	16#4401:
		CreateDriveErrMsgDetails := enumMotorEvents.MotorGeneralError;
		fnLogMsg(ADR(LogMsg_0),LOG_ERROR,'BeckHoff Drive ErrorId %d Starttype not supported',UDINT_TO_DINT(ErrorId),0,0);
	16#4402:
		CreateDriveErrMsgDetails := enumMotorEvents.MotorGeneralError;
		fnLogMsg(ADR(LogMsg_0),LOG_ERROR,'BeckHoff Drive ErrorId %d Command rejected',UDINT_TO_DINT(ErrorId),0,0);
	16#4405:
		CreateDriveErrMsgDetails := enumMotorEvents.MotorGeneralError;
		fnLogMsg(ADR(LogMsg_0),LOG_ERROR,'BeckHoff Drive ErrorId %d Invalid modulo subtype',UDINT_TO_DINT(ErrorId),0,0);
	16#4410:
		CreateDriveErrMsgDetails := enumMotorEvents.MotorGeneralError;
		fnLogMsg(ADR(LogMsg_0),LOG_ERROR,'BeckHoff Drive ErrorId %d Target overrun',UDINT_TO_DINT(ErrorId),0,0);
	16#4411:
		CreateDriveErrMsgDetails := enumMotorEvents.MotorSupplyError;
		fnLogMsg(ADR(LogMsg_0),LOG_ERROR,'BeckHoff Drive ErrorId %d DC-Link undervoltage',UDINT_TO_DINT(ErrorId),0,0);
	16#4412:
 		CreateDriveErrMsgDetails := enumMotorEvents.MotorSupplyError;
		fnLogMsg(ADR(LogMsg_0),LOG_ERROR,'BeckHoff Drive ErrorId %d 2 DC-Link overvoltage',UDINT_TO_DINT(ErrorId),0,0);
	16#4413: 
		CreateDriveErrMsgDetails := enumMotorEvents.MotorSupplyError;
		fnLogMsg(ADR(LogMsg_0),LOG_ERROR,'BeckHoff Drive ErrorId %d I2T Amplifier overload',UDINT_TO_DINT(ErrorId),0,0);
	16#4414:
		CreateDriveErrMsgDetails := enumMotorEvents.MotorSupplyError;
		fnLogMsg(ADR(LogMsg_0),LOG_ERROR,'BeckHoff Drive ErrorId %d I2T Motor overload',UDINT_TO_DINT(ErrorId),0,0);
	16#4415:
		CreateDriveErrMsgDetails := enumMotorEvents.MotorSpeedError;
		fnLogMsg(ADR(LogMsg_0),LOG_ERROR,'BeckHoff Drive ErrorId %d Speed limitation active',UDINT_TO_DINT(ErrorId),0,0);
	16#4416:
		CreateDriveErrMsgDetails := enumMotorEvents.MotorPositionError;
		fnLogMsg(ADR(LogMsg_0),LOG_ERROR,'BeckHoff Drive ErrorId %d Step lost detected',UDINT_TO_DINT(ErrorId),0,0);
	16#8001:
		CreateDriveErrMsgDetails := enumMotorEvents.MotorGeneralError;
		fnLogMsg(ADR(LogMsg_0),LOG_ERROR,'BeckHoff Drive ErrorId %d Error',UDINT_TO_DINT(ErrorId),0,0);
	16#8002:
		CreateDriveErrMsgDetails := enumMotorEvents.DriveComError ;
		fnLogMsg(ADR(LogMsg_0),LOG_ERROR,'BeckHoff Drive ErrorId %d Communication aborted',UDINT_TO_DINT(ErrorId),0,0);

	16#8003:
		CreateDriveErrMsgDetails := enumMotorEvents.PLCIllegalParam;
		fnLogMsg(ADR(LogMsg_0),LOG_ERROR,'BeckHoff Drive ErrorId %d Configuration error',UDINT_TO_DINT(ErrorId),0,0);
	16#8100:
		CreateDriveErrMsgDetails := enumMotorEvents.MotorGeneralError;
		fnLogMsg(ADR(LogMsg_0),LOG_ERROR,'BeckHoff Drive ErrorId %d Status word set',UDINT_TO_DINT(ErrorId),0,0);
	16#8101:
		CreateDriveErrMsgDetails := enumMotorEvents.PLCIllegalParam;
		fnLogMsg(ADR(LogMsg_0),LOG_ERROR,'BeckHoff Drive ErrorId %d Operation mode incompatible to PDO',UDINT_TO_DINT(ErrorId),0,0);
	16#8102:
		CreateDriveErrMsgDetails := enumMotorEvents.PLCIllegalParam;
		fnLogMsg(ADR(LogMsg_0),LOG_ERROR,'BeckHoff Drive ErrorId %d Invalid combination of Inputs and Outputs PDOs',UDINT_TO_DINT(ErrorId),0,0);

	16#8104:
		CreateDriveErrMsgDetails := enumMotorEvents.MotorOverTemp ;
		fnLogMsg(ADR(LogMsg_0),LOG_ERROR,'BeckHoff Drive ErrorId %d Terminal-Overtemperature',UDINT_TO_DINT(ErrorId),0,0);
	
	16#8105:
		CreateDriveErrMsgDetails := enumMotorEvents.MotorGeneralError ;
		fnLogMsg(ADR(LogMsg_0),LOG_ERROR,'BeckHoff Drive ErrorId %d PD-Watchdog',UDINT_TO_DINT(ErrorId),0,0);
	16#8135:
		CreateDriveErrMsgDetails := enumMotorEvents.MotorGeneralError ;
		fnLogMsg(ADR(LogMsg_0),LOG_ERROR,'BeckHoff Drive ErrorId %d Large cycle time',UDINT_TO_DINT(ErrorId),0,0);
	16#8200:
		CreateDriveErrMsgDetails := enumMotorEvents.PLCillegalMsg ;
		fnLogMsg(ADR(LogMsg_0),LOG_ERROR,'BeckHoff Drive ErrorId %d Write access error',UDINT_TO_DINT(ErrorId),0,0);
	16#8201:
		CreateDriveErrMsgDetails := enumMotorEvents.MotorSupplyError ;
		fnLogMsg(ADR(LogMsg_0),LOG_ERROR,'BeckHoff Drive ErrorId %d No com to field-side (Auxiliary voltage missing)',UDINT_TO_DINT(ErrorId),0,0);
	16#82FF:
		CreateDriveErrMsgDetails := enumMotorEvents.MotorGeneralError ;
		fnLogMsg(ADR(LogMsg_0),LOG_ERROR,'BeckHoff Drive ErrorId %d Bootmode not activated',UDINT_TO_DINT(ErrorId),0,0);
	16#8300:
		CreateDriveErrMsgDetails := enumMotorEvents.MotorPositionError ;
		fnLogMsg(ADR(LogMsg_0),LOG_ERROR,'BeckHoff Drive ErrorId %d Set position error',UDINT_TO_DINT(ErrorId),0,0);
	16#8301:
		CreateDriveErrMsgDetails := enumMotorEvents.PLCIllegalParam ;
		fnLogMsg(ADR(LogMsg_0),LOG_ERROR,'BeckHoff Drive ErrorId %d Encoder increments not configured',UDINT_TO_DINT(ErrorId),0,0);
	16#8302:
		CreateDriveErrMsgDetails := enumMotorEvents.MotorFeedBackErr ;
		fnLogMsg(ADR(LogMsg_0),LOG_ERROR,'BeckHoff Drive ErrorId %d Encoder-Error',UDINT_TO_DINT(ErrorId),0,0);

	16#8400:
		CreateDriveErrMsgDetails := enumMotorEvents.PLCIllegalParam;
		fnLogMsg(ADR(LogMsg_0),LOG_ERROR,'BeckHoff Drive ErrorId %d Incorrect drive configuration',UDINT_TO_DINT(ErrorId),0,0);
		
	16#8401:
		CreateDriveErrMsgDetails := enumMotorEvents.MotorSpeedError;
		fnLogMsg(ADR(LogMsg_0),LOG_ERROR,'BeckHoff Drive ErrorId %d Limiting of calibration velocity',UDINT_TO_DINT(ErrorId),0,0);
		
	16#8402:
		CreateDriveErrMsgDetails := enumMotorEvents.DriveNotEnabled;
		fnLogMsg(ADR(LogMsg_0),LOG_ERROR,'BeckHoff Drive ErrorId %d Emergency stop activated',UDINT_TO_DINT(ErrorId),0,0);
	16#8403:
		CreateDriveErrMsgDetails := enumMotorEvents.MotorSupplyError;
		fnLogMsg(ADR(LogMsg_0),LOG_ERROR,'BeckHoff Drive ErrorId %d ADC Error',UDINT_TO_DINT(ErrorId),0,0);
	16#8404:
		CreateDriveErrMsgDetails := enumMotorEvents.MotorSupplyError;
		fnLogMsg(ADR(LogMsg_0),LOG_ERROR,'BeckHoff Drive ErrorId %d Overcurrent',UDINT_TO_DINT(ErrorId),0,0);
	16#8405:
		CreateDriveErrMsgDetails := enumMotorEvents.MotorPositionError;
		fnLogMsg(ADR(LogMsg_0),LOG_ERROR,'BeckHoff Drive ErrorId %d Invalid modulo position',UDINT_TO_DINT(ErrorId),0,0);
	16#8406:
		CreateDriveErrMsgDetails := enumMotorEvents.MotorSupplyError;
		fnLogMsg(ADR(LogMsg_0),LOG_ERROR,'BeckHoff Drive ErrorId %d Undervoltage DC-Link',UDINT_TO_DINT(ErrorId),0,0);
	16#8407:
		CreateDriveErrMsgDetails := enumMotorEvents.MotorSupplyError;
		fnLogMsg(ADR(LogMsg_0),LOG_ERROR,'BeckHoff Drive ErrorId %d Overvoltage DC-Link',UDINT_TO_DINT(ErrorId),0,0);
	16#8408:
		CreateDriveErrMsgDetails := enumMotorEvents.MotorSupplyError;
		fnLogMsg(ADR(LogMsg_0),LOG_ERROR,'BeckHoff Drive ErrorId %d I2T-Model Amplifier overload',UDINT_TO_DINT(ErrorId),0,0);
	16#8409:
		CreateDriveErrMsgDetails := enumMotorEvents.MotorSupplyError;
		fnLogMsg(ADR(LogMsg_0),LOG_ERROR,'BeckHoff Drive ErrorId %d I2T-Model motor overload',UDINT_TO_DINT(ErrorId),0,0);
		
	16#8415:
		CreateDriveErrMsgDetails := enumMotorEvents.PLCIllegalParam;
		fnLogMsg(ADR(LogMsg_0),LOG_ERROR,'BeckHoff Drive ErrorId %d Invalid modulo factor',UDINT_TO_DINT(ErrorId),0,0);
	16#8440:
		CreateDriveErrMsgDetails := enumMotorEvents.MotorSupplyError;
		fnLogMsg(ADR(LogMsg_0),LOG_ERROR,'BeckHoff Drive ErrorId %d Motor cable not connected',UDINT_TO_DINT(ErrorId),0,0);

	ELSE
		fnLogMsg(ADR(LogMsg_0),LOG_ERROR,'unknown BeckHoff Drive ErrorId %d ',UDINT_TO_DINT(ErrorId),0,0);
		CreateDriveErrMsgDetails := enumMotorEvents.NoEvents;
END_CASE
END_METHOD

METHOD DriveErrorHandling : BOOL
VAR_INST
	
	ErrHandleState	: INT;

	SoEReset_FB	: FB_SoEReset;
	EcSoERead_DriveError_FB		: FB_EcSoERead;
	tmpDriveErrId				: UINT;
	NewMsgID					: BYTE;
	PrevMsgID					: BYTE;
	DiagMsg                     : STRING[100];
	EcCoeSdoRead_DriveErrorFB	: FB_EcCoeSdoRead;
	MC_Reset_FB					: MC_Reset;
	tempErrorEntry			    : Eh_ErrorEntry_typ;
	ErrorByte1                  : UINT;
	ErrorByte2                  : UINT;
	BeckHoffLastError       	: UDINT; 
	BeckHoffLastErrorCounter    : UDINT := 0; 
END_VAR


CASE ErrHandleState OF
	0: // logic init
		GetErrCanAdr();	
		ErrHandleState	:= 200;
		
		
	//************************* CAN Logic **********************************************
	200: // wait errors
		{warning disable C0371}
		IF AxisRef.Status.DriveDeviceError OR AxisRef.NcToPlc.ErrorCode = 18000 THEN
			SoEReset_FB.Execute				:= FALSE;
			EcSoERead_DriveError_FB.bExecute	:= FALSE;
			ErrHandleState	:= 210;
		ELSIF AxisRef.NcToPlc.ErrorCode <> 0 
			AND AxisRef.NcToPlc.ErrorCode <> 18000 THEN
			// ETZ Axis.NcToPlc.ErrorCode
			ErrHandleState	:= 300;
		ELSIF AxisCtrlPtr^.Output.Error.fbErrorHandler.EntriesCount > 0 THEN
			// do nothing
		END_IF
		
		IF AxisRef.Status.DriveDeviceError = FALSE THEN
			BeckHoffLastError := 0;
			BeckHoffLastErrorCounter := 0;
		END_IF
		{warning restore C0371}
	210: // wait speed decrease
		IF AxisCtrlPtr^.Output.monitor.ActVelocity < 500 THEN
			ErrHandleState	:= 211;	// read can error
		END_IF
		
	211:// MSG ID read new 
		PrevMsgID := NewMsgID;
		EcCoeSdoRead_DriveErrorFB.sNetId		:= strEcNetId;
		EcCoeSdoRead_DriveErrorFB.nSlaveAddr	:= AxisCtrlPtr^.Input.Parameter.Drive.EtherCatAddr;
		CoeErrIdSubIndex					    := 16#02 ; 			// MSG ID read new 
		EcCoeSdoRead_DriveErrorFB.nIndex		:= CoeErrIdIndex; 
		EcCoeSdoRead_DriveErrorFB.nSubIndex	    := CoeErrIdSubIndex; 
		EcCoeSdoRead_DriveErrorFB.pDstBuf		:= ADR(NewMsgID);
		EcCoeSdoRead_DriveErrorFB.cbBufLen		:= SIZEOF(NewMsgID);
		EcCoeSdoRead_DriveErrorFB.tTimeout		:= T#10S;
		IF NOT EcCoeSdoRead_DriveErrorFB.bBusy THEN
			EcCoeSdoRead_DriveErrorFB.bExecute		:= TRUE;
			
			ErrHandleState	:= 212;
		END_IF	
	212:
		IF NOT EcCoeSdoRead_DriveErrorFB.bBusy THEN
			EcCoeSdoRead_DriveErrorFB.bExecute		:= FALSE;
			IF NOT EcCoeSdoRead_DriveErrorFB.bError THEN				
				
				IF PrevMsgID <> NewMsgID THEN
					// Read Msg
					ErrHandleState	:= 213;
				ELSE
					ErrHandleState	:= 200;	
				END_IF
			ELSE
				fnLogMsg(ADR(LogMsg_0),LOG_ERROR,'NO LINKS FOR DRIVE or Wrong Obj  obj index=%d subindex=%d ErrID %d ',CoeErrIdIndex,CoeErrIdSubIndex,UDINT_TO_DINT(EcCoeSdoRead_DriveErrorFB.nErrId ));
				ErrHandleState	:= 221;	
				DebugError := 1;
			END_IF
		END_IF
	213:
		EcCoeSdoRead_DriveErrorFB.sNetId		:= strEcNetId;
		EcCoeSdoRead_DriveErrorFB.nSlaveAddr	:= AxisCtrlPtr^.Input.Parameter.Drive.EtherCatAddr;
		
		CoeErrIdSubIndex					    := NewMsgID ; 	
		
		EcCoeSdoRead_DriveErrorFB.nIndex		:= CoeErrIdIndex; 
		EcCoeSdoRead_DriveErrorFB.nSubIndex	    := CoeErrIdSubIndex; 
		EcCoeSdoRead_DriveErrorFB.pDstBuf		:= ADR(DiagMsg);
		EcCoeSdoRead_DriveErrorFB.cbBufLen		:= ErrorMSgSize;
		EcCoeSdoRead_DriveErrorFB.tTimeout		:= T#20S;
		IF NOT EcCoeSdoRead_DriveErrorFB.bBusy THEN
			EcCoeSdoRead_DriveErrorFB.bExecute		:= TRUE;
			ErrHandleState	:= 214;	// MC_Reset
		END_IF	
	214:
		IF NOT EcCoeSdoRead_DriveErrorFB.bBusy THEN
			EcCoeSdoRead_DriveErrorFB.bExecute		:= FALSE;
			IF NOT EcCoeSdoRead_DriveErrorFB.bError THEN
				
				ErrHandleState	:= 220;	// Parse error ID
				ErrorByte1 := DiagMsg[6];
				ErrorByte2 := DiagMsg[7]; 
								
				tmpDriveErrId := ErrorByte1 OR SHL(ErrorByte2,8) ;				
				
			ELSE
				fnLogMsg(ADR(LogMsg_0),LOG_ERROR,'St 214 Error read obj index=%d subindex=%d ErrID %d ',CoeErrIdIndex,CoeErrIdSubIndex,TO_DINT(EcCoeSdoRead_DriveErrorFB.nErrId) );
				ErrHandleState	:= 221;	
				
				DebugError := 2;
			END_IF
		END_IF	
	//Parse error ID
	220:
				IF tmpDriveErrId <> 1 THEN
					// Add Drive Error to ErrorHandler
					tmp_ErrorEntry.ErrorId		:= tmpDriveErrId;
		//			IF BeckHoffLastError <>  tmp_ErrorEntry.ErrorId OR BeckHoffLastErrorCounter > 10  THEN
					
						
						tmp_ErrorEntry.ErrorText	:= AxisCtrlPtr^.Input.Parameter.ThreadName;
						tmp_ErrorEntry.ErrorText	:= CONCAT(tmp_ErrorEntry.ErrorText,'Beckhoff Drive ErrorID: ');
						tmp_ErrorEntry.ErrorText	:= CONCAT(tmp_ErrorEntry.ErrorText, UDINT_TO_STRING(tmp_ErrorEntry.ErrorId));
						tmp_ErrorEntry.ErrorText	:= CONCAT(tmp_ErrorEntry.ErrorText, ', Or 0x');
						tmp_ErrorEntry.ErrorText	:= CONCAT(tmp_ErrorEntry.ErrorText, UDINT_TO_HEX_STRING(tmp_ErrorEntry.ErrorId));
						
						tmp_ErrorEntry.MotorEvents  := CreateDriveErrMsgDetails(tmp_ErrorEntry.ErrorId);
						fnLogMsg(ADR(LogMsg_0),LOG_ERROR,tmp_ErrorEntry.ErrorText,0,0,0);
						//ETZ to Add method for Log			
						AxisCtrlPtr^.Output.Error.fbErrorHandler.ErrorPush(tmp_ErrorEntry);
						BeckHoffLastError := tmp_ErrorEntry.ErrorId;
						BeckHoffLastErrorCounter := 0;
			(*		ELSE
						BeckHoffLastErrorCounter := BeckHoffLastErrorCounter + 1;	
					END_IF	*)
				END_IF				
				ErrHandleState	:= 300;	// MC_Reset
		
 	221:
				
					// Add Drive Error to ErrorHandler
					tmp_ErrorEntry.ErrorId		:= 16#8002;
					tmp_ErrorEntry.ErrorText	:= AxisCtrlPtr^.Input.Parameter.ThreadName;
					tmp_ErrorEntry.ErrorText	:= CONCAT(tmp_ErrorEntry.ErrorText,' Drive ErrorID: ');
					tmp_ErrorEntry.ErrorText	:= CONCAT(tmp_ErrorEntry.ErrorText, UDINT_TO_STRING(tmp_ErrorEntry.ErrorId));
					tmp_ErrorEntry.ErrorText	:= CONCAT(tmp_ErrorEntry.ErrorText, ', Or 0x');
					tmp_ErrorEntry.ErrorText	:= CONCAT(tmp_ErrorEntry.ErrorText, UDINT_TO_HEX_STRING(tmp_ErrorEntry.ErrorId));
					
					tmp_ErrorEntry.MotorEvents  := CreateDriveErrMsgDetails(tmp_ErrorEntry.ErrorId);
					fnLogMsg(ADR(LogMsg_0),LOG_ERROR,tmp_ErrorEntry.ErrorText,0,0,0);
					//ETZ to Add method for Log			
					AxisCtrlPtr^.Output.Error.fbErrorHandler.ErrorPush(tmp_ErrorEntry);
								
				ErrHandleState	:= 300;	// MC_Reset
	300: // Run MC_Reset
		MC_Reset_FB.Execute	:= TRUE;
		ErrHandleState		:= 301;
	301:
		{warning disable C0371}
		IF MC_Reset_FB.Done 
			AND AxisRef.NcToPlc.ErrorCode = 0
			(*AND Axis.Status.DriveDeviceError = FALSE*) THEN
			MC_Reset_FB.Execute	:= FALSE;
	
			ErrHandleState	:= 0;
		ELSIF (MC_Reset_FB.Done AND AxisRef.NcToPlc.ErrorCode <> 0) THEN
			
			MC_Reset_FB.Execute	:= FALSE;	
			ErrHandleState		:= 300;	
	
		ELSIF MC_Reset_FB.Error THEN
			MC_Reset_FB.Execute	:= FALSE;
			// Add FB Error to ErrorHandler
			tmp_ErrorEntry.ErrorId		:= MC_Reset_FB.ErrorID;
			tmp_ErrorEntry.ErrorText	:= 'FB MC_Reset_FB ErrorID: ';
			tmp_ErrorEntry.ErrorText	:= CONCAT(tmp_ErrorEntry.ErrorText, UDINT_TO_STRING(tmp_ErrorEntry.ErrorId));
			AxisCtrlPtr^.Output.Error.fbErrorHandler.ErrorPush(tmp_ErrorEntry);
			
			ErrHandleState	:= 0;
		END_IF
		{warning restore C0371}
		IF (AxisCtrlPtr^.Output.Status.CommunicationError = TRUE) THEN
			MC_Reset_FB.Execute	:= FALSE;
			ErrHandleState		:= 400;	
		END_IF
	400:
		IF (AxisCtrlPtr^.Output.Status.CommunicationError = FALSE) THEN
			ErrHandleState	:= 300;	
		END_IF
			

END_CASE

EcSoERead_DriveError_FB();
EcCoeSdoRead_DriveErrorFB();
{warning disable C0371}
SoEReset_FB(Axis:= AxisRef);
MC_Reset_FB(Axis:= AxisRef);
	
{warning restore C0371}
END_METHOD

METHOD GetErrCanAdr : BOOL
VAR_INPUT
END_VAR

CoeErrIdIndex		:= 16#10F3;

		
//CoeErrIdIndex	:= 16#603F;
END_METHOD

END_FUNCTION_BLOCK

// ---- POUs/Lib/Motion/CanOpenAxis/BeckHoff/BeckHoffIntegratedAxis_FB.TcPOU
FUNCTION_BLOCK PUBLIC BeckHoffIntegratedAxis_FB EXTENDS BeckHoffBasicAxis_FB  
VAR_INPUT		
	io_SafetyState: 	BOOL;	
END_VAR

VAR_OUTPUT	
END_VAR

VAR
	 
	
END_VAR


CoEDrive_Ctrl_Adr.DCVoltage.Index 	 := 16#6079; 
CoEDrive_Ctrl_Adr.DCVoltage.SunIndex  := 0;
CoEDrive_Ctrl_Adr.DCVoltage.Size      := 4;

AxisCtrlPtr^.Input.Parameter.Drive.eDriveType := enumDriveType.eIntegratedBeckhoff;	
AxisCtrlPtr^.Input.Parameter.Drive.VendorNameID := eVendorNameID.Beckhoff;
	
 	
SUPER^(AxisRef:=AxisRef);

AxisCtrlPtr^.Output.Status.DriveEnable:=	io_SafetyState;

METHOD GetCanOpenAdr : BOOL
VAR_INPUT
END_VAR
    SUPER^.GetCanOpenAdr();	
	
	
	CoEDrive_Ctrl_Adr.DCVoltage.Index 	 := 16#9010; 
	CoEDrive_Ctrl_Adr.DCVoltage.SunIndex  := 12;
	CoEDrive_Ctrl_Adr.DCVoltage.Size      := 2;
END_METHOD

METHOD HomeLagError : BOOL
VAR_INPUT
	Execute: BOOL;
END_VAR

VAR_INST
	LagErrorState : INT;
	HomingLagErrorTrig: 		Trigger;
	io_TorqueLimitPersent_Mem:	UINT;
	PositionBias:				LREAL;	
END_VAR
Reset:= Execute;
IF HomeTrig.EDGEPOS(Reset) THEN
	Reset:=	FALSE;
	LagErrorState:=1;
	HomingActive:= 	TRUE ;
	AxisCtrlPtr^.Output.Status.MC_Home.Done:= FALSE ;
	fbMC_MoveVel.Execute:= FALSE ;
	fbMC_MoveRel.Execute:= FALSE ;
END_IF

IF Execute THEN
	CASE LagErrorState OF
		
		1:		
			io_TorqueLimitPersent_Mem:=	io_TorqueLimitPersent;							
			io_TorqueLimitPersent:=	AxisCtrlPtr^.Input.Parameter.HomeOptions.stLagErr.TorqueLimitPersent;				
			LagErrorState:= LagErrorState +1;
						 		
		2:	
			IF WriteNC_AxisBoolParam(MC_AxisParameter:=MC_AxisParameter.EnablePosLagMonitoring,ParamValue:=FALSE) THEN
				LagErrorState:= LagErrorState +1;	
			END_IF
																
		3: 										
			IF AxisCtrlPtr^.Input.Parameter.HomeOptions.stBasic.StartDirection = eHomeModeOption.eNEGATIVE THEN								
				fbMC_MoveVel.Direction:= 	MC_Negative_Direction;  					
			ELSIF AxisCtrlPtr^.Input.Parameter.HomeOptions.stBasic.StartDirection = eHomeModeOption.ePOSITIVE THEN								
				fbMC_MoveVel.Direction:= 	MC_Positive_Direction;										
			END_IF
			
			fbMC_MoveVel.Velocity:= AxisCtrlPtr^.Input.Parameter.HomeOptions.stBasic.SwitchVelo;
	
			fbMC_MoveVel.Execute:= 	TRUE ;
			
			LagErrorState:= LagErrorState + 1;
			
		4: 	
			IF (ABS(AxisCtrlPtr^.Output.monitor.ActLagError) > AxisCtrlPtr^.Input.Parameter.HomeOptions.stLagErr.LagErr) THEN
				LagErrorState:= LagErrorState + 1;	
			END_IF
		
		5:	
			IF Stop() THEN
				LagErrorState:= LagErrorState + 2;
				Delay(IN:=	FALSE);					
			END_IF
(*					
		6:	InternalPowerHandle:=	TRUE;
			AxisCtrlPtr^.Input.Command.Power:= FALSE;
			IF AxisCtrlPtr^.Output.Status.AxisStatus.Disabled THEN
				LagErrorState:= LagErrorState + 1;	
			END_IF
*)			
		7:	Delay(IN:=	TRUE,PT:=T#1S);		
			IF Delay.Q THEN
				Delay(IN:=FALSE);	
				LagErrorState:= LagErrorState +2;
			END_IF
(*	
		8:	InternalPowerHandle:=	FALSE;
			AxisCtrlPtr^.Input.Command.Power:= TRUE;
			
			IF (AxisCtrlPtr^.Output.Status.AxisStatus.Disabled = FALSE) THEN
				
				io_TorqueLimitPersent:=	io_TorqueLimitPersent_Mem;	
				LagErrorState:= LagErrorState + 1;	
			END_IF
*)						
		9: 	io_TorqueLimitPersent:=	io_TorqueLimitPersent_Mem;	
			IF AxisCtrlPtr^.Input.Parameter.HomeOptions.stBasic.StartDirection = eHomeModeOption.eNEGATIVE THEN													
				fbMC_MoveRel.Distance:=		AxisCtrlPtr^.Input.Parameter.HomeOptions.stLagErr.TriggerOffsetPos ;					
			ELSIF AxisCtrlPtr^.Input.Parameter.HomeOptions.stBasic.StartDirection = eHomeModeOption.ePOSITIVE THEN								
				fbMC_MoveRel.Distance:=		AxisCtrlPtr^.Input.Parameter.HomeOptions.stLagErr.TriggerOffsetPos*(-1) ;											
			END_IF
			fbMC_MoveRel.Velocity:= AxisCtrlPtr^.Input.Parameter.HomeOptions.stBasic.TriggerVelo;
			
			fbMC_MoveRel.Execute:= 	TRUE ;
			LagErrorState:= LagErrorState + 1;
	 		
					
		10:	
			IF fbMC_MoveRel.Done THEN
				AxisCtrlPtr^.Output.monitor.stAbsEncoder.BlockOffsetPosition := AxisCtrlPtr^.Output.monitor.ActPosition ;
				(*				
				fbMC_Home.HomingMode:= 	MC_Direct ;
				fbMC_Home.Position:= 	(AxisCtrlPtr^.Input.Parameter.HomeOptions.stBasic.HomeSetPos); 
				fbMC_Home.Execute:= 	TRUE;
				LagErrorState:= LagErrorState + 1;*)
				LagErrorState:= 100;
			END_IF
			
		11:	IF fbMC_Home.Done THEN			
				fbMC_Home.Execute:= 	FALSE;
				LagErrorState:= 100;	
			END_IF
																				
		100:			
			AxisCtrlPtr^.Input.Command.Home:= FALSE ;
			HomingActive:= 				FALSE;
			fbMC_Home.Execute:= 		FALSE;
			AxisCtrlPtr^.Output.Status.MC_Home.Done:= TRUE ;
			HomeLagError:=	TRUE;
			LagErrorState:= 0;		
	END_CASE

END_IF
 
			
fbMC_MoveVel.Acceleration  	:= AxisCtrlPtr^.Input.Parameter.HomeOptions.stBasic.Acc;  
fbMC_MoveVel.Deceleration  	:= AxisCtrlPtr^.Input.Parameter.HomeOptions.stBasic.Dcc;  
fbMC_MoveVel.Jerk			:= AxisCtrlPtr^.Input.Parameter.HomeOptions.stBasic.Jerk;
fbMC_MoveVel.Options		:= AxisCtrlPtr^.Input.Parameter.Options;
fbMC_MoveVel.BufferMode		:= AxisCtrlPtr^.Input.Parameter.BufferMode;

fbMC_MoveRel.Acceleration  	:= AxisCtrlPtr^.Input.Parameter.HomeOptions.stBasic.Acc; 
fbMC_MoveRel.Deceleration  	:= AxisCtrlPtr^.Input.Parameter.HomeOptions.stBasic.Dcc;
fbMC_MoveRel.Jerk			:= AxisCtrlPtr^.Input.Parameter.HomeOptions.stBasic.Jerk;
fbMC_MoveRel.Options		:= AxisCtrlPtr^.Input.Parameter.Options;
fbMC_MoveRel.BufferMode		:= AxisCtrlPtr^.Input.Parameter.BufferMode;

{warning disable C0371}
//Warning: Access to VAR_IN_OUT <Var> declared in <POU> from external context <Method/Transition/Property>

fbMC_Home(Axis:= AxisRef);	
fbMC_MoveVel(Axis:= AxisRef);
fbMC_MoveRel(Axis:= AxisRef);

fbMC_Stop.Deceleration:= 	AxisCtrlPtr^.Input.Parameter.Deceleration;
fbMC_Stop.Jerk:=			AxisCtrlPtr^.Input.Parameter.Jerk;
fbMC_Stop.Options:= 		AxisCtrlPtr^.Input.Parameter.Options;
fbMC_Stop(Axis := AxisRef) ;
{warning restore C0371}

THIS^.HomingGlobalHandle();
END_METHOD

METHOD ReadActualTorque : LREAL
VAR_INPUT
END_VAR
VAR_INST
		
END_VAR


// Units [rms]

{warning disable C0371}
IF AxisCtrlPtr^.Output.Status.Drive.ActiveHW THEN
	AxisCtrlPtr^.Output.monitor.ActualTorque	:=  ( -(AxisRef.NcToPlc.ActTorque) / 100.0) * AxisCtrlPtr^.Input.Parameter.Ratedtorque;
ELSE
	AxisCtrlPtr^.Output.monitor.ActualTorque	:=  ((THIS^.io_ActualTorque) / 1000.0) * AxisCtrlPtr^.Input.Parameter.Ratedtorque;
END_IF	

{warning restore C0371}
END_METHOD

END_FUNCTION_BLOCK

// ---- POUs/Lib/Motion/CanOpenAxis/BeckHoff/bk5xxxBasicAxis_FB.TcPOU
FUNCTION_BLOCK bk5xxxBasicAxis_FB EXTENDS BeckHoffBasicAxis_FB
VAR_INPUT
	pDigIn: 	POINTER TO INT;	
END_VAR
VAR_OUTPUT
END_VAR
VAR
	
END_VAR


AxisCtrlPtr^.Input.Parameter.Drive.eDriveType	:= enumDriveType.e5xxxBeckhoff;
AxisCtrlPtr^.Input.Parameter.Drive.VendorNameID	:= eVendorNameID.Beckhoff;


SUPER^(AxisRef:=AxisRef);

IF (pDigIn <> 0) THEN
	AxisCtrlPtr^.Output.Status.DriveEnable	:= pDigIn^.7;
ELSE
	AxisCtrlPtr^.Output.Status.DriveEnable	:= TRUE;
END_IF

END_FUNCTION_BLOCK

// ---- POUs/Lib/Motion/CanOpenAxis/BeckHoff/el7xxxBasicAxis_FB.TcPOU
FUNCTION_BLOCK el7xxxBasicAxis_FB EXTENDS BeckHoffBasicAxis_FB
VAR_INPUT
	pDigIn: 	POINTER TO INT;	
END_VAR
VAR_OUTPUT
END_VAR
VAR
	
END_VAR


AxisCtrlPtr^.Input.Parameter.Drive.eDriveType := enumDriveType.eEL70xx;
AxisCtrlPtr^.Input.Parameter.Drive.VendorNameID := eVendorNameID.Beckhoff;


SUPER^(AxisRef:=AxisRef);

IF (pDigIn <> 0) THEN
	AxisCtrlPtr^.Output.Status.DriveEnable	:= pDigIn^.7;
ELSE
	AxisCtrlPtr^.Output.Status.DriveEnable	:= TRUE;
END_IF

METHOD HomeLagErrExternFeedBack : BOOL
VAR_INPUT
	Execute: BOOL;
END_VAR

VAR_INST
	fbEcCoeSdoWriteMaxCurrent	: FB_EcCoeSdoWrite;
	State:INT;	
	ExtLagErrPrevState : INT;
	HomeTrig: Trigger;
	Reset:BOOL;	
	Delay:	TON;	
	LastActExternEncodPos:		UDINT;
	DiffExternEncodPos:			DINT;
	LatchSetPos:				LREAL;			
	CalckedLagError:			LREAL;
	EncdSampleTimer:			TON;
	StartPosMonitor:			BOOL;
		
END_VAR
Reset:= Execute;
IF HomeTrig.EDGEPOS(Reset) THEN
	Reset:=	FALSE;
	State:=1;
	
	HomeLagErrExternFeedBack:= FALSE ;
	HomingActive:= 	TRUE ;
	AxisCtrlPtr^.Output.Status.MC_Home.Done:= FALSE ;
	fbMC_MoveVel.Execute:= FALSE ;
	fbMC_MoveRel.Execute:= FALSE ;
END_IF

IF Execute THEN
	CASE State OF
		
		1:									
			fbEcCoeSdoWriteMaxCurrent.sNetId:= 		strEcNetId;
			fbEcCoeSdoWriteMaxCurrent.nSlaveAddr:= 	AxisCtrlPtr^.Input.Parameter.Drive.EtherCatAddr;
			fbEcCoeSdoWriteMaxCurrent.nSubIndex:=	1;
			fbEcCoeSdoWriteMaxCurrent.nIndex:= 		16#8010;  			
			fbEcCoeSdoWriteMaxCurrent.pSrcBuf:=		 ADR(AxisCtrlPtr^.Input.Parameter.HomeOptions.stLagErr.BlockSearchMaxCurrent); 
			fbEcCoeSdoWriteMaxCurrent.cbBufLen:= 	SIZEOF(AxisCtrlPtr^.Input.Parameter.HomeOptions.stLagErr.BlockSearchMaxCurrent); 
			fbEcCoeSdoWriteMaxCurrent.bExecute:= 	TRUE; 
			fbEcCoeSdoWriteMaxCurrent.tTimeout:= 	T#2S;					
			State:= State +1;							
			 
		2:		
			IF NOT fbEcCoeSdoWriteMaxCurrent.bBusy THEN
				fbEcCoeSdoWriteMaxCurrent.bExecute:= FALSE;
				IF NOT fbEcCoeSdoWriteMaxCurrent.bError THEN																									
					State:= State +1;
				ELSE
					fbEcCoeSdoWriteMaxCurrent.bExecute:= FALSE;
					fnLogMsg(ADR(LogMsg_0),LOG_ERROR,Concat('ADS Error Code %d: ',F_ADStoStr(fbEcCoeSdoWriteMaxCurrent.nErrId)),UDINT_TO_DINT(fbEcCoeSdoWriteMaxCurrent.nErrId),0,0);
					State:= 0;				
				END_IF				
			END_IF 		 
		3:	
			IF WriteNC_AxisBoolParam(MC_AxisParameter:=MC_AxisParameter.EnablePosLagMonitoring,ParamValue:=FALSE) THEN
				State:= State +1;	
			END_IF
						
										
		4: 										
			IF AxisCtrlPtr^.Input.Parameter.HomeOptions.stBasic.StartDirection = eHomeModeOption.eNEGATIVE THEN								
				fbMC_MoveVel.Direction:= 	MC_Negative_Direction; 					
			ELSIF AxisCtrlPtr^.Input.Parameter.HomeOptions.stBasic.StartDirection = eHomeModeOption.ePOSITIVE THEN								
				fbMC_MoveVel.Direction:= 	MC_Positive_Direction;										
			END_IF
			
			fbMC_MoveVel.Velocity:= AxisCtrlPtr^.Input.Parameter.HomeOptions.stBasic.SwitchVelo;			
			fbMC_MoveVel.Execute:= 	TRUE ;
			LastActExternEncodPos:=	AxisCtrlPtr^.Output.monitor.ActExternEncodPos;						
			State:= State + 1;
			
		5:	IF AxisCtrlPtr^.Output.Status.AxisStatus.ContinuousMotion THEN
				EncdSampleTimer(IN:= NOT(EncdSampleTimer.Q),PT:=T#0.2S);
				IF EncdSampleTimer.Q THEN	
					State:= State + 1;
				END_IF	
			END_IF
		6: 							
			DiffExternEncodPos:=ABS(UDINT_TO_DINT(AxisCtrlPtr^.Output.monitor.ActExternEncodPos) - UDINT_TO_DINT(LastActExternEncodPos));
			IF DiffExternEncodPos <= 4 THEN
				LatchSetPos:=	AxisCtrlPtr^.Output.monitor.ActPosition;			
				State:= State + 1;
			ELSE
				LastActExternEncodPos:=	AxisCtrlPtr^.Output.monitor.ActExternEncodPos;	
				State:= 5;
			END_IF			
					
		7:									
			CalckedLagError:=	ABS(AxisCtrlPtr^.Output.monitor.ActPosition - LatchSetPos);										
			IF (CalckedLagError > AxisCtrlPtr^.Input.Parameter.HomeOptions.stLagErr.LagErr) THEN
				State:= State + 1;	
			END_IF
			
		
		8:	
			IF Stop() THEN
				State:= State + 1;				
			END_IF
					
		9:	InternalPowerHandle:=	TRUE;
			AxisCtrlPtr^.Input.Command.Power:= FALSE;
			IF AxisCtrlPtr^.Output.Status.AxisStatus.Disabled THEN
				State:= State + 1;	
			END_IF
			
		10:	Delay(IN:=	TRUE,PT:=T#0.5S);		
			IF Delay.Q THEN
				Delay(IN:=FALSE);	
				State:= State +1;
			END_IF
			
		11:	InternalPowerHandle:=	FALSE;
			AxisCtrlPtr^.Input.Command.Power:= TRUE;
			State:= State +1;
		
		12:	
	
			IF (AxisCtrlPtr^.Output.Status.MC_Power.Status = TRUE) THEN
				State:= State + 1;	
			END_IF
			
			
		13:	Delay(IN:=	TRUE,PT:=T#0.5S);		
			IF Delay.Q THEN
				Delay(IN:=FALSE);
					
				State:= State +1;
			END_IF
			
		14:		
		

			IF fbEcCoeSdoWriteMaxCurrent.bBusy = FALSE THEN
				fbEcCoeSdoWriteMaxCurrent.sNetId:= 		strEcNetId;
				fbEcCoeSdoWriteMaxCurrent.nSlaveAddr:= 	AxisCtrlPtr^.Input.Parameter.Drive.EtherCatAddr;
				fbEcCoeSdoWriteMaxCurrent.nSubIndex:=	1;
				fbEcCoeSdoWriteMaxCurrent.nIndex:= 		16#8010;  				
				fbEcCoeSdoWriteMaxCurrent.pSrcBuf:=		 ADR(AxisCtrlPtr^.Input.Parameter.HomeOptions.stLagErr.BlockExitMaxCurrent); 				
				fbEcCoeSdoWriteMaxCurrent.cbBufLen:= 	SIZEOF(AxisCtrlPtr^.Input.Parameter.HomeOptions.stLagErr.BlockExitMaxCurrent); 
				fbEcCoeSdoWriteMaxCurrent.bExecute:= 	TRUE; 
				fbEcCoeSdoWriteMaxCurrent.tTimeout:= 	T#2S;	
								
				
				State:= State +1;				
			END_IF
			
			
			
							
		15:		
			State:= State +1;
		16:	
			IF NOT fbEcCoeSdoWriteMaxCurrent.bBusy THEN
				fbEcCoeSdoWriteMaxCurrent.bExecute:= FALSE;
				IF NOT fbEcCoeSdoWriteMaxCurrent.bError THEN																									
					State:= State +1;
				ELSE
					fbEcCoeSdoWriteMaxCurrent.bExecute:= FALSE;
					fnLogMsg(ADR(LogMsg_0),LOG_ERROR,Concat('ADS Error Code %d: ',F_ADStoStr(fbEcCoeSdoWriteMaxCurrent.nErrId)),UDINT_TO_DINT(fbEcCoeSdoWriteMaxCurrent.nErrId),0,0);
					State:= 0;				
				END_IF				
			END_IF 		 
				
		17:	
			IF WriteNC_AxisBoolParam(MC_AxisParameter:=MC_AxisParameter.EnablePosLagMonitoring,ParamValue:=FALSE) THEN			
				State:= State +1;	
			END_IF	
			
														
		18:		
			fbMC_Home.HomingMode:= 	MC_Direct ;
			fbMC_Home.Position:= 	0;
			fbMC_Home.Execute:= 	TRUE;	
			State:= State + 1;
							
		19:	
			IF fbMC_Home.Done THEN
				fbMC_Home.Execute := FALSE;		
				IF AxisCtrlPtr^.Input.Parameter.HomeOptions.stBasic.StartDirection = eHomeModeOption.eNEGATIVE THEN													
					fbMC_MoveRel.Distance:=		AxisCtrlPtr^.Input.Parameter.HomeOptions.stLagErr.TriggerOffsetPos ;					
				ELSIF AxisCtrlPtr^.Input.Parameter.HomeOptions.stBasic.StartDirection = eHomeModeOption.ePOSITIVE THEN								
					fbMC_MoveRel.Distance:=		AxisCtrlPtr^.Input.Parameter.HomeOptions.stLagErr.TriggerOffsetPos*(-1) ;											
				END_IF
				fbMC_MoveRel.Velocity:= AxisCtrlPtr^.Input.Parameter.HomeOptions.stBasic.TriggerVelo;
				
				fbMC_MoveRel.Execute:= 	TRUE ;
				State:= State + 1;	
			END_IF
			
		20:	IF fbMC_MoveRel.Done THEN
				fbMC_MoveRel.Execute := FALSE;
				fbMC_Home.HomingMode:= 	MC_Direct ;
				//fbMC_Home.Options:= 	AxisCtrlPtr^.Input.Parameter.HomeOptions.NcHomeOption;
				fbMC_Home.Position:= 	(AxisCtrlPtr^.Input.Parameter.HomeOptions.stBasic.HomeSetPos) * (-1); 
				fbMC_Home.Execute:= 	TRUE;	
				State := 100 ;
			END_IF
																											
		100:
			IF fbMC_Home.Done THEN
				AxisCtrlPtr^.Input.Command.Home:= FALSE ;
				HomingActive:= 							FALSE;
				HomeLagErrExternFeedBack:= 		TRUE;
				fbMC_Home.Execute:= 					FALSE;
				AxisCtrlPtr^.Output.Status.MC_Home.Done:= TRUE ;
				State:= 0;
			END_IF
	END_CASE
	IF ExtLagErrPrevState <> State THEN
		fnLogMsg(ADR(LogMsg_0),LOG_INFO,'Drive Lag Err step %d',State,0,0);
		ExtLagErrPrevState := State;
	END_IF	
	
END_IF
 

fbMC_MoveVel.Acceleration  	:= AxisCtrlPtr^.Input.Parameter.Acceleration;
fbMC_MoveVel.Deceleration  	:= AxisCtrlPtr^.Input.Parameter.Deceleration;
fbMC_MoveVel.Jerk			:= AxisCtrlPtr^.Input.Parameter.Jerk;
fbMC_MoveVel.Options		:= AxisCtrlPtr^.Input.Parameter.Options;
fbMC_MoveVel.BufferMode		:= AxisCtrlPtr^.Input.Parameter.BufferMode;

fbMC_MoveRel.Acceleration  	:= AxisCtrlPtr^.Input.Parameter.Acceleration;
fbMC_MoveRel.Deceleration  	:= AxisCtrlPtr^.Input.Parameter.Deceleration;
fbMC_MoveRel.Jerk			:= AxisCtrlPtr^.Input.Parameter.Jerk;
fbMC_MoveRel.Options		:= AxisCtrlPtr^.Input.Parameter.Options;
fbMC_MoveRel.BufferMode		:= AxisCtrlPtr^.Input.Parameter.BufferMode;

{warning disable C0371}
//Warning: Access to VAR_IN_OUT <Var> declared in <POU> from external context <Method/Transition/Property>
fbMC_Home(Axis:= AxisRef);	
fbMC_MoveVel(Axis:= AxisRef);
fbMC_MoveRel(Axis:= AxisRef);


fbMC_Stop.Deceleration:= 	AxisCtrlPtr^.Input.Parameter.Deceleration;
fbMC_Stop.Jerk:=			AxisCtrlPtr^.Input.Parameter.Jerk;
fbMC_Stop.Options:= 		AxisCtrlPtr^.Input.Parameter.Options;
fbMC_Stop(Axis := AxisRef) ;
{warning restore C0371}

fbEcCoeSdoWriteMaxCurrent();

THIS^.HomingGlobalHandle();
END_METHOD

METHOD HomeLagErrInternalEnc : BOOL
VAR_INPUT
	Execute: BOOL;
END_VAR

VAR_INST
	fbEcCoeSdoWriteMaxCurrent	: FB_EcCoeSdoWrite;
//	State:INT;	
//	HomeTrig: Trigger;
//	Reset:BOOL;	
//	Delay:	TON;	
END_VAR
Reset:= Execute;
IF HomeTrig.EDGEPOS(Reset) THEN
	Reset:=	FALSE;
	State:=1;
	HomeLagErrInternalEnc:= FALSE ;
	HomingActive:= 	TRUE ;
	AxisCtrlPtr^.Output.Status.MC_Home.Done:= FALSE ;
	fbMC_MoveVel.Execute:= FALSE ;
	fbMC_MoveRel.Execute:= FALSE ;
END_IF

IF Execute THEN
	CASE State OF
		
		1:									
			fbEcCoeSdoWriteMaxCurrent.sNetId:= 		strEcNetId;
			fbEcCoeSdoWriteMaxCurrent.nSlaveAddr:= 	AxisCtrlPtr^.Input.Parameter.Drive.EtherCatAddr;
			fbEcCoeSdoWriteMaxCurrent.nSubIndex:=	1;
			fbEcCoeSdoWriteMaxCurrent.nIndex:= 		16#8010;  
			fbEcCoeSdoWriteMaxCurrent.pSrcBuf:=		 ADR(AxisCtrlPtr^.Input.Parameter.HomeOptions.stLagErr.BlockSearchMaxCurrent); 
			fbEcCoeSdoWriteMaxCurrent.cbBufLen:= 	SIZEOF(AxisCtrlPtr^.Input.Parameter.HomeOptions.stLagErr.BlockSearchMaxCurrent); 
			fbEcCoeSdoWriteMaxCurrent.bExecute:= 	TRUE; 
			fbEcCoeSdoWriteMaxCurrent.tTimeout:= 	T#2S;					
			State:= State +1;
				
			//IF (NOT SDOrw.Output.Status.EcCoeSdoWrite.bError) THEN
			//	SDOrw.Input.Command.EcCoeSdoWrite.Enable:= TRUE;
			//END_IF
			//SDOrw.Input.Parameter.EcCoeSdoWrite.sNetId 		:= strEcNetId;
		    //SDOrw.Input.Parameter.EcCoeSdoWrite.nSlaveAddr	:= AxisCtrlPtr^.Input.Parameter.nSlaveAddr;
			//SDOrw.Input.Parameter.EcCoeSdoWrite.nIndex		:= 	16#8010;	
		    //SDOrw.Input.Parameter.EcCoeSdoWrite.nSubIndex	:= 	1; 			
			//SDOrw.Input.Parameter.EcCoeSdoWrite.pSrcBuf		:=  ADR(AxisCtrlPtr^.Input.Parameter.HomeOptions.BlockSearchMaxCurrent); 
			//SDOrw.Input.Parameter.EcCoeSdoWrite.cbBufLen	:=  SIZEOF(AxisCtrlPtr^.Input.Parameter.HomeOptions.BlockSearchMaxCurrent);		
			//State:= State +1;
			 
		2:
			//IF THIS^.EcCoeSdoWrite() THEN 
			//	 State:= State +1;
			// END_IF	
			IF NOT fbEcCoeSdoWriteMaxCurrent.bBusy THEN
				fbEcCoeSdoWriteMaxCurrent.bExecute:= FALSE;
				IF NOT fbEcCoeSdoWriteMaxCurrent.bError THEN																									
					State:= State +1;
				ELSE
					fbEcCoeSdoWriteMaxCurrent.bExecute:= FALSE;
					fnLogMsg(ADR(LogMsg_0),LOG_ERROR,Concat('int ADS Error Code %d index-0x8010: ',F_ADStoStr(fbEcCoeSdoWriteMaxCurrent.nErrId)),UDINT_TO_DINT(fbEcCoeSdoWriteMaxCurrent.nErrId),0,0);
					State:= 0;				
				END_IF				
			END_IF 		 
		3:	
			IF WriteNC_AxisBoolParam(MC_AxisParameter:=MC_AxisParameter.EnablePosLagMonitoring,ParamValue:=FALSE) THEN
				State:= State +1;	
			END_IF
						
										
		4: 										
			IF AxisCtrlPtr^.Input.Parameter.HomeOptions.stBasic.StartDirection = eHomeModeOption.eNEGATIVE THEN								
				fbMC_MoveVel.Direction:= 	MC_Negative_Direction; 					
			ELSIF AxisCtrlPtr^.Input.Parameter.HomeOptions.stBasic.StartDirection = eHomeModeOption.ePOSITIVE THEN								
				fbMC_MoveVel.Direction:= 	MC_Positive_Direction;										
			END_IF
			
			fbMC_MoveVel.Velocity:= AxisCtrlPtr^.Input.Parameter.HomeOptions.stBasic.SwitchVelo;
	
			fbMC_MoveVel.Execute:= 	TRUE ;
			
			State:= State + 1;
			
		5: 	
			IF (ABS(AxisCtrlPtr^.Output.monitor.ActLagError) > AxisCtrlPtr^.Input.Parameter.HomeOptions.stLagErr.LagErr) THEN
				State:= State + 1;	
			END_IF
		
		6:	
			IF Stop() THEN
				State:= State + 1;				
			END_IF
					
		7:	InternalPowerHandle:=	TRUE;
			AxisCtrlPtr^.Input.Command.Power:= FALSE;
			IF AxisCtrlPtr^.Output.Status.AxisStatus.Disabled THEN
				State:= State + 1;	
			END_IF
			
		8:	Delay(IN:=	TRUE,PT:=T#1S);		
			IF Delay.Q THEN
				Delay(IN:=FALSE);	
				State:= State +1;
			END_IF
			
		9:	InternalPowerHandle:=	FALSE;
			AxisCtrlPtr^.Input.Command.Power:= TRUE;
			IF (AxisCtrlPtr^.Output.Status.AxisStatus.Disabled = FALSE) THEN
				State:= State + 1;	
			END_IF
			
			
		10:	
		(*
			IF (NOT SDOrw.Output.Status.EcCoeSdoWrite.bError) THEN
				SDOrw.Input.Command.EcCoeSdoWrite.Enable 		:= TRUE;
			END_IF
			SDOrw.Input.Parameter.EcCoeSdoWrite.sNetId 		:= strEcNetId;
		    SDOrw.Input.Parameter.EcCoeSdoWrite.nSlaveAddr	:= LREAL_TO_UINT(AxisCtrlPtr^.Input.Parameter.Drive.EtherCatAddr.Value);
			SDOrw.Input.Parameter.EcCoeSdoWrite.nIndex		:= 	16#8010;	
		    SDOrw.Input.Parameter.EcCoeSdoWrite.nSubIndex	:= 	1; 			
			SDOrw.Input.Parameter.EcCoeSdoWrite.pSrcBuf		:=  ADR(AxisCtrlPtr^.Input.Parameter.HomeOptions.stLagErr.BlockExitMaxCurrent); 
			SDOrw.Input.Parameter.EcCoeSdoWrite.cbBufLen	:=  SIZEOF(AxisCtrlPtr^.Input.Parameter.HomeOptions.stLagErr.BlockExitMaxCurrent);	
		*)
			
			fbEcCoeSdoWriteMaxCurrent.sNetId:= 		strEcNetId;
			fbEcCoeSdoWriteMaxCurrent.nSlaveAddr:= AxisCtrlPtr^.Input.Parameter.Drive.EtherCatAddr;
			fbEcCoeSdoWriteMaxCurrent.nSubIndex:= 1;
			fbEcCoeSdoWriteMaxCurrent.nIndex:= 		16#8010;
			fbEcCoeSdoWriteMaxCurrent.pSrcBuf:=		ADR(AxisCtrlPtr^.Input.Parameter.HomeOptions.stLagErr.BlockExitMaxCurrent); 
			fbEcCoeSdoWriteMaxCurrent.cbBufLen:= SIZEOF(AxisCtrlPtr^.Input.Parameter.HomeOptions.stLagErr.BlockExitMaxCurrent);
			fbEcCoeSdoWriteMaxCurrent.bExecute:=  TRUE;
			fbEcCoeSdoWriteMaxCurrent.tTimeout:= T#2S;
			
			State:= State +1; 

		11:	
			IF NOT fbEcCoeSdoWriteMaxCurrent.bBusy THEN
				fbEcCoeSdoWriteMaxCurrent.bExecute:= FALSE;		
				 State:= State +1;
			END_IF		
				
		12:	
			IF WriteNC_AxisBoolParam(MC_AxisParameter:=MC_AxisParameter.EnablePosLagMonitoring,ParamValue:=TRUE) THEN			
				State:= State +1;	
			END_IF	
			
														
		13:		
			fbMC_Home.HomingMode:= 	MC_Direct ;
			//fbMC_Home.Options:= 	AxisCtrlPtr^.Input.Parameter.HomeOptions.NcHomeOption ;
			fbMC_Home.Position:= 	0;
			fbMC_Home.Execute:= 	TRUE;	
			State:= State + 1;
							
		14:	
			IF fbMC_Home.Done THEN
				fbMC_Home.Execute := FALSE;		
				IF AxisCtrlPtr^.Input.Parameter.HomeOptions.stBasic.StartDirection = eHomeModeOption.eNEGATIVE THEN													
					fbMC_MoveRel.Distance:=		AxisCtrlPtr^.Input.Parameter.HomeOptions.stLagErr.TriggerOffsetPos ;					
				ELSIF AxisCtrlPtr^.Input.Parameter.HomeOptions.stBasic.StartDirection = eHomeModeOption.ePOSITIVE THEN								
					fbMC_MoveRel.Distance:=		AxisCtrlPtr^.Input.Parameter.HomeOptions.stLagErr.TriggerOffsetPos*(-1) ;											
				END_IF
				fbMC_MoveRel.Velocity:= AxisCtrlPtr^.Input.Parameter.HomeOptions.stBasic.TriggerVelo;
				
				fbMC_MoveRel.Execute:= 	TRUE ;
				State:= State + 1;	
			END_IF
			
		15:	IF fbMC_MoveRel.Done THEN
				fbMC_Home.HomingMode:= 	MC_Direct ;
				//fbMC_Home.Options:= 	AxisCtrlPtr^.Input.Parameter.HomeOptions.NcHomeOption;
				fbMC_Home.Position:= 	(AxisCtrlPtr^.Input.Parameter.HomeOptions.stBasic.HomeSetPos) * (-1); 
				fbMC_Home.Execute:= 	TRUE;	
				State := 100 ;
			END_IF
																											
		100:
			IF fbMC_Home.Done THEN
				AxisCtrlPtr^.Input.Command.Home:= FALSE ;
				HomingActive:= 				FALSE;
				HomeLagErrInternalEnc:= 		TRUE;
				fbMC_Home.Execute:= 		FALSE;
				AxisCtrlPtr^.Output.Status.MC_Home.Done:= TRUE ;
				State:= 0;
			END_IF
	END_CASE

END_IF
 

fbMC_MoveVel.Acceleration  	:= AxisCtrlPtr^.Input.Parameter.Acceleration;
fbMC_MoveVel.Deceleration  	:= AxisCtrlPtr^.Input.Parameter.Deceleration;
fbMC_MoveVel.Jerk			:= AxisCtrlPtr^.Input.Parameter.Jerk;
fbMC_MoveVel.Options		:= AxisCtrlPtr^.Input.Parameter.Options;
fbMC_MoveVel.BufferMode		:= AxisCtrlPtr^.Input.Parameter.BufferMode;

fbMC_MoveRel.Acceleration  	:= AxisCtrlPtr^.Input.Parameter.Acceleration;
fbMC_MoveRel.Deceleration  	:= AxisCtrlPtr^.Input.Parameter.Deceleration;
fbMC_MoveRel.Jerk			:= AxisCtrlPtr^.Input.Parameter.Jerk;
fbMC_MoveRel.Options		:= AxisCtrlPtr^.Input.Parameter.Options;
fbMC_MoveRel.BufferMode		:= AxisCtrlPtr^.Input.Parameter.BufferMode;

{warning disable C0371}
//Warning: Access to VAR_IN_OUT <Var> declared in <POU> from external context <Method/Transition/Property>

fbMC_Home(Axis:= AxisRef);	
fbMC_MoveVel(Axis:= AxisRef);
fbMC_MoveRel(Axis:= AxisRef);

fbMC_Stop.Deceleration:= 	AxisCtrlPtr^.Input.Parameter.Deceleration;
fbMC_Stop.Jerk:=			AxisCtrlPtr^.Input.Parameter.Jerk;
fbMC_Stop.Options:= 		AxisCtrlPtr^.Input.Parameter.Options;
fbMC_Stop(Axis := AxisRef) ;
{warning restore C0371}
fbEcCoeSdoWriteMaxCurrent();

THIS^.HomingGlobalHandle();
END_METHOD

METHOD HomeLagError : BOOL
VAR_INPUT
	Execute: BOOL;
END_VAR

VAR_INST
	LagErrorState : INT;
	HomingLagErrorTrig: Trigger;
END_VAR
VAR
	
END_VAR


IF HomingLagErrorTrig.EDGEPOS(Execute) THEN
	LagErrorState := 1;
	HomeLagError := FALSE;
END_IF


IF HomingLagErrorTrig.EDGENEG(Execute) THEN
	
	LagErrorState := 0;
	
END_IF

CASE LagErrorState OF
	 
	
	1:
		HomeLagErrExternFeedBack(FALSE);
		HomeLagErrInternalEnc(FALSE);
		LagErrorState := LagErrorState +1;
	2:
		IF AxisCtrlPtr^.Input.Parameter.HomeOptions.stBasic.ExternalEncoder THEN
			IF HomeLagErrExternFeedBack(TRUE) THEN
				LagErrorState := LagErrorState +1;				
			END_IF
		ELSE
			IF HomeLagErrInternalEnc(TRUE) THEN
				LagErrorState := LagErrorState +1;				
			END_IF
	
		END_IF		
	3:
		HomeLagError := TRUE;
	
END_CASE
END_METHOD

END_FUNCTION_BLOCK

// ---- POUs/Lib/Motion/CanOpenAxis/BeckHoff/ep7xxxBasicAxis_FB.TcPOU
FUNCTION_BLOCK ep7xxxBasicAxis_FB EXTENDS BeckHoffBasicAxis_FB
VAR_INPUT
	rDriveEnable: 	REFERENCE TO BOOL; // Reference to external drive enable signal
END_VAR
VAR_OUTPUT
END_VAR
VAR
	
END_VAR


AxisCtrlPtr^.Input.Parameter.Drive.eDriveType	:= enumDriveType.eEP70xx;
AxisCtrlPtr^.Input.Parameter.Drive.VendorNameID	:= eVendorNameID.Beckhoff;

SUPER^(AxisRef:=AxisRef);

IF __ISVALIDREF(rDriveEnable) THEN
	AxisCtrlPtr^.Output.Status.DriveEnable	:= rDriveEnable;
ELSE
	AxisCtrlPtr^.Output.Status.DriveEnable	:= TRUE;
END_IF

END_FUNCTION_BLOCK

// ---- POUs/Lib/Motion/CanOpenAxis/Elmo/ElmoVelocityCtrlAxis_FB.TcPOU
FUNCTION_BLOCK PUBLIC ElmoVelocityCtrlAxis_FB EXTENDS VelocityCtrlAxis_FB  
VAR_INPUT
	

END_VAR

VAR_OUTPUT
END_VAR
	
VAR

	
END_VAR

SUPER^();

METHOD METH_ChangeToVelMode : BOOL
VAR_INPUT
	Execute : BOOL;
END_VAR
IF InitSctrlTrigger.EDGEPOS( Execute) THEN
	CngToVelocityState := 1;
	METH_ChangeToVelMode := FALSE;
	rAxisBasicFB.AxisCtrlPtr^.Input.Command.Power := FALSE;
	
	OldCyclicTorque := 0;		
	OldSctrlKp 		:= 0;
	OldSctrlKi 		:= 0;			
	rAxisBasicFB.Meth_WriteObj (FALSE, enumMotionobject.OPERATION_MODE, TO_LREAL(eDriveModeOfOperation.CyclicSyncVelocity));

END_IF

IF InitSctrlTrigger.EDGENEG( Execute) THEN
	CngToVelocityState := 0;
END_IF


CASE CngToVelocityState OF
	0:
		METH_ChangeToVelMode := FALSE;
	1:
		IF ReadPosCtrlParamDone = FALSE THEN
			 Meth_ReadPosCtrlValues(FALSE);
			 CngToVelocityState := CngToVelocityState +1;	
		ELSE
			CngToVelocityState := CngToVelocityState +2;
		END_IF		
	2:
		IF Meth_ReadPosCtrlValues(TRUE) THEN
			
			rAxisBasicFB.Meth_WriteObj (FALSE, enumMotionobject.OPERATION_MODE,eDriveModeOfOperation.CyclicSyncVelocity);
			
			CngToVelocityState := CngToVelocityState +1;
			
		END_IF
	3:	//Change mode to velocity control
		IF rAxisBasicFB.Meth_WriteObj (TRUE, enumMotionobject.OPERATION_MODE,eDriveModeOfOperation.CyclicSyncVelocity) THEN			
			rAxisBasicFB.Meth_WriteObj (FALSE, enumMotionobject.OPERATION_MODE,eDriveModeOfOperation.CyclicSyncVelocity);
			CngToVelocityState := CngToVelocityState +1;
		END_IF
		
	4://Disable Gain Control
		IF NOT rAxisBasicFB.AxisCtrlPtr^.Output.Status.MC_Power.Status THEN
			IF rAxisBasicFB.Meth_WriteObj (TRUE, enumMotionobject.GAIN_SCHEDULE,0) THEN			
				rAxisBasicFB.Meth_WriteObj (FALSE, enumMotionobject.OPERATION_MODE,eDriveModeOfOperation.CyclicSyncVelocity);			
				CngToVelocityState := CngToVelocityState +1;
			END_IF
		END_IF	
	
	5:	
		rAxisBasicFB.AxisCtrlPtr^.Input.Command.Power := TRUE;
		IF rAxisBasicFB.AxisCtrlPtr^.Output.Status.AxisStatus.StandStill THEN
			CngToVelocityState := CngToVelocityState +1;
		END_IF
	6:
		IF  rAxisBasicFB.Meth_WriteObj(TRUE, enumMotionObject.ACC_CLOSE_POS_ERR ,   rVelocityCtrl.Input.Parameter.CyclicVelocity    , Error =>Error ) THEN
			rAxisBasicFB.Meth_WriteObj(FALSE, enumMotionObject.ACC_CLOSE_POS_ERR ,0 );
			CngToVelocityState := CngToVelocityState +1;
		END_IF	
	
	7:	
		METH_ChangeToVelMode := TRUE;
END_CASE
END_METHOD

METHOD Meth_InitSctrl : BOOL
VAR_INPUT
	Execute : BOOL;
END_VAR


VAR_OUTPUT
	Error : BOOL;
END_VAR
IF InitSctrlTrigger.EDGEPOS(Execute) THEN
	InitSctrlState  := 1;
	Meth_InitSctrl := FALSE;
	rAxisBasicFB.Meth_InitVelKP (FALSE,0);
	rAxisBasicFB.Meth_InitVelKI(FALSE,0);
	Error := FALSE;
END_IF


IF InitSctrlTrigger.EDGENEG(Execute) THEN
	
	 InitSctrlState:= 0;
END_IF


CASE InitSctrlState OF
 
		
	1:
		 			
	 
	 	IF rAxisBasicFB.Meth_InitVelKP (TRUE,(rVelocityCtrl.Input.Parameter.SctrlKp), Error=>Error) THEN
	 		OldSctrlKp := rVelocityCtrl.Input.Parameter.SctrlKp;
	 		InitSctrlState := InitSctrlState +1;
	 		rAxisBasicFB.Meth_InitVelKP (FALSE,rVelocityCtrl.Input.Parameter.SctrlKp);
	 	END_IF	
 	  
			

	2:
	
			IF rAxisBasicFB.Meth_InitVelKI(TRUE,(rVelocityCtrl.Input.Parameter.SctrlKi), Error=>Error) THEN
				rAxisBasicFB.Meth_InitVelKP (FALSE,rVelocityCtrl.Input.Parameter.SctrlKi);
				OldSctrlKi := rVelocityCtrl.Input.Parameter.SctrlKi ;
				InitSctrlState := InitSctrlState +1;
			END_IF	

		IF Error THEN
		//	
		END_IF
		
	3:		
		rVelocityCtrl.Output.Status.SctrlInitialized := TRUE;
		Meth_InitSctrl := TRUE; 
	END_CASE
END_METHOD

METHOD Meth_ReadPosCtrlValues : BOOL
VAR_INPUT
	Execute : BOOL;
END_VAR


VAR_INST
	// Service Functions Variablea
	ReadPosCtrlTrigger : Trigger ;
	ReadPosCtrlState   : SINT;
END_VAR	

VAR_OUTPUT
	Error : BOOL;	
END_VAR
IF ReadPosCtrlTrigger.EDGEPOS(Execute) THEN
	ReadPosCtrlState  := 1;
	Meth_ReadPosCtrlValues := FALSE;
	Error := FALSE;
	rAxisBasicFB.Meth_ReadObj(FALSE, enumMotionObject.MAX_TORQUE, Value =>rVelocityCtrl.Output.monitor.OrgMaxTorque, Error =>Error );
END_IF


IF ReadPosCtrlTrigger.EDGENEG(Execute) THEN
	 rAxisBasicFB.Meth_ReadObj(FALSE, enumMotionObject.MAX_TORQUE, Value =>rVelocityCtrl.Output.monitor.OrgMaxTorque, Error =>Error );
	 ReadPosCtrlState:= 0;
END_IF


CASE ReadPosCtrlState OF
 
	1:
		IF  rAxisBasicFB.Meth_ReadObj(TRUE, enumMotionObject.TORQUE_OFFSET, Value =>rVelocityCtrl.Output.monitor.OrgCyclicTorque, Error =>Error ) THEN
			rAxisBasicFB.Meth_ReadObj(FALSE, enumMotionObject.TORQUE_OFFSET  );
 			ReadPosCtrlState := ReadPosCtrlState +1;
			Error := FALSE;						
		END_IF
		IF Error THEN
			ReadPosCtrlState := 33;
		END_IF
			
	2:
		IF  rAxisBasicFB.Meth_ReadObj(TRUE, enumMotionObject.VEL_KP, Value =>rVelocityCtrl.Output.monitor.OrgSctrlKp, Error =>Error ) THEN
			rVelocityCtrl.Output.monitor.OrgVelKp := rVelocityCtrl.Output.monitor.OrgSctrlKp;
			rAxisBasicFB.Meth_ReadObj(FALSE, enumMotionObject.TORQUE_OFFSET  );
 			ReadPosCtrlState := ReadPosCtrlState +1;
		END_IF
	3:
		IF  rAxisBasicFB.Meth_ReadObj(TRUE, enumMotionObject.VEL_KI, Value =>rVelocityCtrl.Output.monitor.OrgSctrlKi, Error =>Error ) THEN
			rAxisBasicFB.Meth_ReadObj(FALSE, enumMotionObject.TORQUE_OFFSET  );
 			ReadPosCtrlState := ReadPosCtrlState +1;
		END_IF
	
	4:
		IF rAxisBasicFB.Meth_ReadObj (TRUE, enumMotionobject.GAIN_SCHEDULE, Value =>rVelocityCtrl.Output.monitor.OrgGainCtrl, Error =>Error) THEN			
				rAxisBasicFB.Meth_ReadObj(FALSE, enumMotionObject.TORQUE_OFFSET  );
				ReadPosCtrlState := ReadPosCtrlState +1;						
		END_IF		
		
	5:
			IF rAxisBasicFB.Meth_ReadObj (TRUE, enumMotionobject.ACC_CLOSE_POS_ERR, Value =>rVelocityCtrl.Output.monitor.OrgAccToCloseThePosError, Error =>Error) THEN			
				rAxisBasicFB.Meth_ReadObj(FALSE, enumMotionObject.TORQUE_OFFSET  );
				ReadPosCtrlState := ReadPosCtrlState +1;						
			END_IF	
	6:	
		IF rAxisBasicFB.Meth_ReadObj (TRUE, enumMotionobject.MAX_TORQUE  , Value =>rVelocityCtrl.Output.monitor.OrgMaxTorque, Error =>Error) THEN	
				fnLogMsg(ADR(LogMsg_0),LOG_INFO,'MAX_TORQUE org=%d',TO_DINT(rVelocityCtrl.Output.monitor.OrgMaxTorque),0,0);		
				rAxisBasicFB.Meth_ReadObj(FALSE, enumMotionObject.TORQUE_OFFSET  );
				ReadPosCtrlState := ReadPosCtrlState +1;						
		 	END_IF		

	7:
	
				
		ReadPosCtrlParamDone := TRUE;
		Meth_ReadPosCtrlValues := TRUE; 
	END_CASE
END_METHOD

METHOD Meth_ReturnOrgPosCtrlValues : BOOL
VAR_INPUT
	Execute : BOOL;
END_VAR


VAR_INST
		// Service Functions Variablea
	ReturnOrgTrigger : Trigger ;
	ReturnOrgState   : SINT;
END_VAR	

VAR_OUTPUT
	Error : BOOL;
END_VAR
IF ReturnOrgTrigger.EDGEPOS(Execute) THEN
	ReturnOrgState  := 1;
	Meth_ReturnOrgPosCtrlValues := FALSE;
	Error := FALSE;
	rAxisBasicFB.Meth_WriteObj(FALSE, enumMotionObject.MAX_TORQUE, rVelocityCtrl.Output.monitor.OrgMaxTorque, Error =>Error );
END_IF


IF ReturnOrgTrigger.EDGENEG(Execute) THEN
	 rAxisBasicFB.Meth_WriteObj(FALSE, enumMotionObject.MAX_TORQUE,  rVelocityCtrl.Output.monitor.OrgMaxTorque, Error =>Error );
	 ReturnOrgState:= 0;
END_IF


CASE ReturnOrgState OF
 
		
	1:	
		IF  rAxisBasicFB.Meth_WriteObj(TRUE, enumMotionObject.GAIN_SCHEDULE,  rVelocityCtrl.Output.monitor.OrgGainCtrl, Error =>Error ) THEN
			rAxisBasicFB.Meth_WriteObj(FALSE, enumMotionObject.GAIN_SCHEDULE ,0 );
 			ReturnOrgState := ReturnOrgState +1;
		END_IF		
			
	2:
		IF  rAxisBasicFB.Meth_WriteObj(TRUE, enumMotionObject.VEL_KP,  rVelocityCtrl.Output.monitor.OrgSctrlKp, Error =>Error ) THEN
			rAxisBasicFB.Meth_WriteObj(FALSE,enumMotionObject.VEL_KP,0  );
 			ReturnOrgState := ReturnOrgState +1;
		END_IF
	3:
		IF  rAxisBasicFB.Meth_WriteObj(TRUE, enumMotionObject.VEL_KI,  rVelocityCtrl.Output.monitor.OrgSctrlKi, Error =>Error ) THEN
			rAxisBasicFB.Meth_WriteObj(FALSE, enumMotionObject.VEL_KP ,0 );
 			ReturnOrgState := ReturnOrgState +1;
		END_IF
	
	4:
		IF  rAxisBasicFB.Meth_WriteObj(TRUE, enumMotionObject.TORQUE_OFFSET, rVelocityCtrl.Output.monitor.OrgCyclicTorque , Error =>Error ) THEN
			rAxisBasicFB.Meth_WriteObj(FALSE, enumMotionObject.VEL_KP ,0 );
 			ReturnOrgState := ReturnOrgState +1;
		END_IF
		
	5:				
		IF  rAxisBasicFB.Meth_WriteObj(TRUE, enumMotionObject.MAX_TORQUE, rVelocityCtrl.Output.monitor.OrgMaxTorque  , Error =>Error ) THEN
			rAxisBasicFB.Meth_WriteObj(FALSE, enumMotionObject.VEL_KP ,0 );
 			ReturnOrgState := ReturnOrgState +1;
		END_IF
	6:	
		ReadPosCtrlParamDone := TRUE;
		Meth_ReturnOrgPosCtrlValues := TRUE; 
	END_CASE
END_METHOD

END_FUNCTION_BLOCK

// ---- POUs/Lib/Motion/VelocityCtrlAxis_FB.TcPOU
FUNCTION_BLOCK PUBLIC VelocityCtrlAxis_FB
VAR_INPUT
	
	rAxisBasicFB 		: REFERENCE TO BasicAxis_FB ;
	rVelocityCtrl	 	: REFERENCE TO VelocityCtrl_typ ;
		
END_VAR

VAR_OUTPUT
END_VAR
	
VAR
	LogMsgInit		: BOOL;
	LogMsg_0 		: LogMsg ;
	
//	GetCycleTime:	FB_CTRL_GET_TASK_CYCLETIME;
//	CycleTime:		TIME;
//	CycleTimeInit:	BOOL;
	
	
	fbGetCurTaskIdx: 		GETCURTASKINDEX;
    TaskCycleTimeUDINT: 	UDINT;
    TaskCycleTime: 			TIME;

	EnableTrigger : Trigger ;
	
	DisableTriger	: Trigger ;
	Disable			: BOOL ;
	
// Change Oper params
	ChangeModeTrigger   : Trigger ;
	CngToVelocityState 	: SINT;
	PrevCngToVelocityState : SINT;
	// Change Oper params
	InitSctrlTrigger : Trigger ;
	InitSctrlState 	 : SINT;	

	
	ErrorTrig : Trigger ;
	AxisStep     : eVelocityCtrlState ;
	ReturnToAxisStep     : eVelocityCtrlState ;
	
	LastAxisStep : eVelocityCtrlState ;
	
	tmp_ErrorEntry			: Eh_ErrorEntry_typ;
	
	
	
	ReadPosCtrlParamDone 	: BOOL;	
	OldCyclicTorque 		: LREAL;		
	OldSctrlKp 				: LREAL;
	OldSctrlKi 				: LREAL;
	PrevVel 				: LREAL;
	Error					: BOOL;
	//Paramter
		
	CyclicTorqueAtPositionCtrl : LREAL;	
	

	
	Delay 			:	 TON;
	
	StartTestRead: BOOL;
	TestRead : BOOL;
END_VAR

// 
// At default set default torque
//
// Change mode to velocity control
// 
//
//
//
//
IF __ISVALIDREF( rAxisBasicFB) AND __ISVALIDREF(rVelocityCtrl) THEN
	
	

IF NOT LogMsgInit THEN 
	LogMsg_0.logData.category:=	rAxisBasicFB.AxisCtrlPtr^.Input.Parameter.ThreadName;     
	LogMsg_0.Enable:= 	TRUE; 	
END_IF

IF (TaskCycleTimeUDINT = 0) THEN
	fbGetCurTaskIdx();
	TaskCycleTimeUDINT := _TaskInfo[fbGetCurTaskIdx.index].CycleTime;
	TaskCycleTime	:= UDINT_TO_TIME(TaskCycleTimeUDINT/10000); 
END_IF



LogMsg_0.ptrGlobalArray:= 	ADR(LogGlobalArray);
LogMsg_0.ptrEncoderAngle:= 	ADR(rAxisBasicFB.AxisCtrlPtr^.Input.Parameter.PosForLog);



//in case of Stop go to STATE_WAIT
IF (rVelocityCtrl.Output.Status.Active)AND(NOT rVelocityCtrl.Output.Status.InStopVelCtrl)  THEN
	
	
	IF rAxisBasicFB.AxisCtrlPtr^.Output.Status.FAULT THEN
 
			AxisStep := eVelocityCtrlState.VELOCITY_CTRL_STATE_ERROR;	

	ELSIF (rAxisBasicFB.AxisCtrlPtr^.Input.Command.Halt) OR rVelocityCtrl.Input.Command.Stop THEN
		rVelocityCtrl.Input.Command.Stop := FALSE;
		Meth_stop(FALSE);
		AxisStep := eVelocityCtrlState.VELOCITY_CTRL_STATE_STOP ;

		
	ELSIF (rAxisBasicFB.AxisCtrlPtr^.Input.Command.Stop)  THEN 
		AxisStep := eVelocityCtrlState.VELOCITY_CTRL_ACTIVE_STAND_STILL;
		PrevVel :=  rVelocityCtrl.Input.Parameter.CyclicVelocity := 0;
	END_IF	
	
END_IF


IF EnableTrigger.EDGEPOS(rVelocityCtrl.Input.Command.Enable) THEN
 	IF (NOT rVelocityCtrl.Output.Status.Active) AND AxisStep = eVelocityCtrlState.VELOCITY_CTRL_STATE_READY THEN
		METH_ChangeToVelMode(FALSE);
		AxisStep := VELOCITY_CTRL_CNG_TO_VEL_MODE ;
	END_IF	
		
END_IF		
	
IF EnableTrigger.EDGENEG( rVelocityCtrl.Input.Command.Enable) THEN
	IF (rVelocityCtrl.Output.Status.Active) THEN
 		Meth_ExitVelCtrl(FALSE);
		AxisStep :=  eVelocityCtrlState.VELOCITY_CTRL_DISABLE;
	END_IF	
	
END_IF		



CASE AxisStep OF
		
	(******************** WAIT *************************)
		
	VELOCITY_CTRL_STATE_WAIT:	
		rVelocityCtrl.Output.Status.Active := FALSE;
		IF rAxisBasicFB.AxisCtrlPtr^.Output.Status.AxisInitDone
			 THEN
			AxisStep := VELOCITY_CTRL_STATE_READY ;
		END_IF
		
		THIS^.ResetAll_MC_FB();
		
	VELOCITY_CTRL_STATE_READY:
	
		rVelocityCtrl.Output.Status.Active := FALSE;
		IF rVelocityCtrl.Input.Command.InitSctrl THEN
				
				rVelocityCtrl.Input.Command.InitSctrl := FALSE;
				rVelocityCtrl.Output.Status.SctrlInitialized := FALSE;
				Meth_InitSctrl(FALSE);
				
				rAxisBasicFB.Meth_WriteObj(FALSE,enumMotionObject.VEL_KI,0);
				AxisStep :=VELOCITY_CTRL_InitSctrl;
				ReturnToAxisStep := VELOCITY_CTRL_STATE_READY;
 								
		ELSIF rVelocityCtrl.Input.Command.Stop THEN
			
			rVelocityCtrl.Input.Command.Stop  := FALSE;
			AxisStep := VELOCITY_CTRL_STATE_STOP ;
			
		ELSIF rVelocityCtrl.Input.Parameter.CyclicTorque <> OldCyclicTorque THEN
				
				Error := FALSE;
				ReturnToAxisStep := VELOCITY_CTRL_STATE_READY;
				AxisStep :=VELOCITY_CTRL_CHANGE_TORQUE;
				
				rAxisBasicFB.Meth_CngTorqueOffset(FALSE,0);
				rAxisBasicFB.Meth_CngMaxTorque(FALSE,0);
				ReturnToAxisStep := VELOCITY_CTRL_STATE_READY;
				rAxisBasicFB.Meth_WriteObj(FALSE,enumMotionObject.VEL_KI,0);	
				rVelocityCtrl.Output.Status.UpdateTorqueDone := FALSE;		
		END_IF
		

//ReadPosCtrlParamDone
		
	VELOCITY_CTRL_CNG_TO_VEL_MODE:
		// Change mode to velocity control
		IF METH_ChangeToVelMode(TRUE) THEN
			rVelocityCtrl.Output.Status.Active := TRUE;
			AxisStep :=VELOCITY_CTRL_MOVE_VELOCITY;
		END_IF	
			
	VELOCITY_CTRL_READ_POS_CTRL_VALUES:
			IF Meth_ReadPosCtrlValues(TRUE) THEN
				AxisStep :=VELOCITY_CTRL_MOVE_VELOCITY;
			END_IF
	
				
	VELOCITY_CTRL_MOVE_VELOCITY:
	
		IF rVelocityCtrl.Input.Parameter.CyclicVelocity <>0 OR rAxisBasicFB.AxisCtrlPtr^.Output.monitor.ActVelocity <>0  THEN
			Meth_MoveVel();
			AxisStep := VELOCITY_CTRL_WAIT_MOVE_VELOCITY_DONE;
		ELSE
			AxisStep := VELOCITY_CTRL_ACTIVE;
		END_IF	
	
	
	VELOCITY_CTRL_WAIT_MOVE_VELOCITY_DONE:	
		IF rAxisBasicFB.AxisCtrlPtr^.Output.Status.MC_MoveVelocity.In_Velocity THEN
			IF rVelocityCtrl.Input.Parameter.CyclicTorque <> 0 THEN
				Error := FALSE;
				ReturnToAxisStep := VELOCITY_CTRL_ACTIVE;
				AxisStep :=VELOCITY_CTRL_CHANGE_TORQUE;
				rAxisBasicFB.Meth_CngTorqueOffset(FALSE,0);
				rAxisBasicFB.Meth_CngMaxTorque(FALSE,0);
				ReturnToAxisStep := VELOCITY_CTRL_ACTIVE;
				rAxisBasicFB.Meth_WriteObj(FALSE,enumMotionObject.VEL_KI,0);
			ELSE
				PrevVel := rVelocityCtrl.Input.Parameter.CyclicVelocity;
				AxisStep := VELOCITY_CTRL_ACTIVE;
			END_IF	 
	END_IF
		
		
	VELOCITY_CTRL_ACTIVE:
	
			rVelocityCtrl.Output.Status.Active := TRUE;
			IF rVelocityCtrl.Input.Command.Stop THEN
				meth_Stop(FALSE);
				rVelocityCtrl.Input.Command.Stop  := FALSE;
				AxisStep := VELOCITY_CTRL_STATE_STOP ;
				
			ELSIF rVelocityCtrl.Input.Command.InitSctrl THEN
				
				rVelocityCtrl.Input.Command.InitSctrl := FALSE;
				rVelocityCtrl.Output.Status.SctrlInitialized := FALSE;
				Meth_InitSctrl(FALSE);
				
				rAxisBasicFB.Meth_WriteObj(FALSE,enumMotionObject.VEL_KI,0);
				AxisStep :=VELOCITY_CTRL_InitSctrl;
				ReturnToAxisStep := VELOCITY_CTRL_ACTIVE;
				
			ELSIF rVelocityCtrl.Input.Parameter.CyclicTorque <> OldCyclicTorque THEN
				
				Error := FALSE;
				ReturnToAxisStep := VELOCITY_CTRL_ACTIVE;
				AxisStep :=VELOCITY_CTRL_CHANGE_TORQUE;
				rAxisBasicFB.Meth_CngTorqueOffset(FALSE,0);
				rAxisBasicFB.Meth_CngMaxTorque(FALSE,0);
				ReturnToAxisStep := VELOCITY_CTRL_ACTIVE;
				rAxisBasicFB.Meth_WriteObj(FALSE,enumMotionObject.VEL_KI,0);				
			ELSIF rVelocityCtrl.Input.Parameter.CyclicVelocity <> rAxisBasicFB.AxisCtrlPtr^.Input.Parameter.Velocity THEN
					AxisStep := VELOCITY_CTRL_MOVE_VELOCITY;
		 	
			ELSIF rVelocityCtrl.Input.Parameter.CyclicVelocity <> PrevVel THEN
				
				AxisStep := VELOCITY_CTRL_MOVE_VELOCITY;
				
			END_IF	
			
	VELOCITY_CTRL_ACTIVE_STAND_STILL:
			rVelocityCtrl.Output.Status.Active := TRUE;
 			
			IF rVelocityCtrl.Input.Parameter.CyclicVelocity <> PrevVel THEN
				
				AxisStep := VELOCITY_CTRL_MOVE_VELOCITY;
			
			
			ELSIF rVelocityCtrl.Input.Command.InitSctrl THEN
				
				rVelocityCtrl.Input.Command.InitSctrl := FALSE;
				rVelocityCtrl.Output.Status.SctrlInitialized := FALSE;
				Meth_InitSctrl(FALSE);
				
				rAxisBasicFB.Meth_WriteObj(FALSE,enumMotionObject.VEL_KI,0);
				AxisStep :=VELOCITY_CTRL_InitSctrl;
				ReturnToAxisStep := VELOCITY_CTRL_ACTIVE_STAND_STILL;
				
			ELSIF rVelocityCtrl.Input.Parameter.CyclicTorque <> OldCyclicTorque THEN
				
				Error := FALSE;
				ReturnToAxisStep := VELOCITY_CTRL_ACTIVE;
				AxisStep :=VELOCITY_CTRL_CHANGE_TORQUE;
				rAxisBasicFB.Meth_CngTorqueOffset(FALSE,0);
				rAxisBasicFB.Meth_CngMaxTorque(FALSE,0);
				ReturnToAxisStep := VELOCITY_CTRL_ACTIVE_STAND_STILL;
				rAxisBasicFB.Meth_WriteObj(FALSE,enumMotionObject.VEL_KI,0);

		 	
			ELSIF rAxisBasicFB.AxisCtrlPtr^.Output.Status.AxisStatus.Coupled THEN
				IF rAxisBasicFB.AxisCtrlPtr^.Output.monitor.ActVelocity <> 0 THEN
					AxisStep := VELOCITY_CTRL_ACTIVE;
				END_IF 
			END_IF	

	VELOCITY_CTRL_InitSctrl:
	
			IF Meth_InitSctrl(TRUE,Error=>Error) THEN
				AxisStep :=ReturnToAxisStep;			
			END_IF
			
			IF Error THEN
			//	
			END_IF
	VELOCITY_CTRL_CHANGE_TORQUE:	
				
			IF rVelocityCtrl.Input.Parameter.TorqueMode = eTorqueMode.mcFF THEN
				//IF rAxisBasicFB.Meth_CngTorqueOffset(TRUE,rVelocityCtrl.Input.Parameter.CyclicTorque, Error => Error ) THEN
				IF  rAxisBasicFB.Meth_WriteObj(TRUE, enumMotionObject.TORQUE_OFFSET,rVelocityCtrl.Input.Parameter.CyclicTorque, Error => Error ) THEN
					fnLogMsg(ADR(LogMsg_0),LOG_INFO,'Vel Ctrl Change Torque to=%d',LREAL_TO_DINT(rVelocityCtrl.Input.Parameter.CyclicTorque*1000),0,0);
					
					OldCyclicTorque := rVelocityCtrl.Input.Parameter.CyclicTorque;
					rAxisBasicFB.Meth_CngTorqueOffset(FALSE,rVelocityCtrl.Input.Parameter.CyclicTorque);
					AxisStep :=ReturnToAxisStep;	
					rVelocityCtrl.Output.monitor.SetCyclicTorque := rVelocityCtrl.Input.Parameter.CyclicTorque ;
				END_IF							
			
			ELSIF rVelocityCtrl.Input.Parameter.TorqueMode = eTorqueMode.mcLimit THEN
				//IF rAxisBasicFB.Meth_CngMaxTorque(TRUE,rVelocityCtrl.Input.Parameter.CyclicTorque , Error => Error) THEN
				IF  rAxisBasicFB.Meth_WriteObj(TRUE, enumMotionObject.MAX_TORQUE,rVelocityCtrl.Input.Parameter.CyclicTorque, Error => Error ) THEN					
					OldCyclicTorque := rVelocityCtrl.Input.Parameter.CyclicTorque;
					rVelocityCtrl.Output.monitor.SetCyclicTorque := rVelocityCtrl.Input.Parameter.CyclicTorque ;
					rVelocityCtrl.Output.Status.UpdateTorqueDone := TRUE;
					AxisStep :=ReturnToAxisStep;
	
				END_IF
			END_IF
			
	eVelocityCtrlState.VELOCITY_CTRL_STATE_STOP:
		IF Meth_stop(TRUE) THEN
			
			PrevVel :=  rVelocityCtrl.Input.Parameter.CyclicVelocity := 0;
			AxisStep := eVelocityCtrlState.VELOCITY_CTRL_ACTIVE_STAND_STILL;
		END_IF
	
	
	eVelocityCtrlState.VELOCITY_CTRL_DISABLE:
		rVelocityCtrl.Output.Status.InStopVelCtrl := TRUE;
		IF Meth_ExitVelCtrl(TRUE) THEN
			rVelocityCtrl.Output.Status.InStopVelCtrl := FALSE;
			AxisStep := eVelocityCtrlState.VELOCITY_CTRL_STATE_READY;
		END_IF
	eVelocityCtrlState.VELOCITY_CTRL_STATE_RETURN_ORG_VALUES:
		IF Meth_ReturnOrgPosCtrlValues(TRUE) THEN				
			AxisStep := ReturnToAxisStep ;
		END_IF
		
	eVelocityCtrlState.VELOCITY_CTRL_STATE_ERROR:
			rVelocityCtrl.Output.Status.InStopVelCtrl := TRUE;
			IF Meth_ExitVelCtrl(TRUE) THEN			
				rVelocityCtrl.Output.Status.InStopVelCtrl := FALSE;
				AxisStep := eVelocityCtrlState.VELOCITY_CTRL_STATE_WAIT;
			END_IF

			

	
	
END_CASE 



//=====================================================================================================================\\

//IF CyclicAxisCtrlPtr^.Output.Error.ErrorID <> 0 THEN		
	//BasicAxisCtrlPtr^.Output.Error.ErrorID := CyclicAxisCtrlPtr^.Output.Error.ErrorID ;
	//CyclicAxisCtrlPtr^.Output.Error.ErrorID := 0;
//END_IF

	IF LastAxisStep <> AxisStep THEN
		
		fnLogMsg(ADR(LogMsg_0),LOG_INFO,'Vel Ctrl CurSt=%d LstSt=%d',AxisStep,LastAxisStep,0);
		LastAxisStep := AxisStep ;
	END_IF	
	
	IF StartTestRead THEN
		StartTestRead := FALSE;
		Meth_ReadPosCtrlValues(FALSE);
		TestRead := TRUE;
		
	ELSIF TestRead THEN
		IF Meth_ReadPosCtrlValues(TRUE) THEN
			TestRead := FALSE;
		END_IF	
		
	END_IF

	
	
//fnLogTransfer FUNCTION call
fnLogTransfer(ADR(LogMsg_0));
		

END_IF

METHOD AddNCError : BOOL
VAR_INPUT
	ErrorId			: UDINT;
	ErrorPrefix     : STRING[100];
END_VAR

	tmp_ErrorEntry.ErrorId		:= ErrorId;

	tmp_ErrorEntry.ErrorText	:= ErrorPrefix;

	tmp_ErrorEntry.ErrorText	:= CONCAT(tmp_ErrorEntry.ErrorText, UDINT_TO_STRING(tmp_ErrorEntry.ErrorId));
	tmp_ErrorEntry.ErrorText	:= CONCAT(tmp_ErrorEntry.ErrorText, 'Task: ');
	tmp_ErrorEntry.ErrorText	:= CONCAT(tmp_ErrorEntry.ErrorText, rVelocityCtrl.Input.Parameter.ThreadName);	
	tmp_ErrorEntry.ErrorText	:= CONCAT(tmp_ErrorEntry.ErrorText, FC_NcErrorMsg(tmp_ErrorEntry.ErrorId));	
	fnLogMsg(ADR(LogMsg_0),LOG_ERROR,tmp_ErrorEntry.ErrorText,0,0,0);	
	
	tmp_ErrorEntry.MotorEvents := CreateNCErrMsgDetails(tmp_ErrorEntry.ErrorId);
	
	rAxisBasicFB.AxisCtrlPtr^.Output.Error.fbErrorHandler.ErrorPush(tmp_ErrorEntry);
END_METHOD

METHOD METH_ChangeToVelMode : BOOL
VAR_INPUT
	Execute : BOOL;
END_VAR
VAR_INST
	DelayBeforeChangimeMode: TON;
END_VAR
IF InitSctrlTrigger.EDGEPOS( Execute) THEN
	CngToVelocityState := 1;
	METH_ChangeToVelMode := FALSE;
	rAxisBasicFB.AxisCtrlPtr^.Input.Command.Power := FALSE;
	
	OldCyclicTorque := 0;		
	OldSctrlKp 		:= 0;
	OldSctrlKi 		:= 0;			
	rAxisBasicFB.Meth_WriteObj (FALSE, enumMotionobject.OPERATION_MODE,DINT_TO_LREAL(eDriveModeOfOperation.CyclicSyncVelocity));

END_IF

IF InitSctrlTrigger.EDGENEG( Execute) THEN
	CngToVelocityState := 0;
END_IF


CASE CngToVelocityState OF
	0:
		METH_ChangeToVelMode := FALSE;
		 
	1:
		DelayBeforeChangimeMode.IN := FALSE;
		IF ReadPosCtrlParamDone = FALSE THEN
			 Meth_ReadPosCtrlValues(FALSE);
			 CngToVelocityState := CngToVelocityState +1;	
		ELSE
			CngToVelocityState := CngToVelocityState +2;
		END_IF		
	2:
		IF Meth_ReadPosCtrlValues(TRUE) THEN
			
			rAxisBasicFB.Meth_WriteObj (FALSE, enumMotionobject.OPERATION_MODE,eDriveModeOfOperation.CyclicSyncVelocity);
			
			CngToVelocityState := CngToVelocityState +1;
			
		END_IF
	3:	//Change mode to velocity control
		IF rAxisBasicFB.Meth_WriteObj (TRUE, enumMotionobject.OPERATION_MODE,eDriveModeOfOperation.CyclicSyncVelocity) THEN			
			rAxisBasicFB.Meth_WriteObj (FALSE, enumMotionobject.OPERATION_MODE,eDriveModeOfOperation.CyclicSyncVelocity);
			CngToVelocityState := CngToVelocityState +1;
		END_IF
		
	4://Disable Gain Control
		IF NOT rAxisBasicFB.AxisCtrlPtr^.Output.Status.MC_Power.Status THEN
			IF rAxisBasicFB.Meth_WriteObj (TRUE, enumMotionobject.GAIN_SCHEDULE,0) THEN			
				rAxisBasicFB.Meth_WriteObj (FALSE, enumMotionobject.OPERATION_MODE,eDriveModeOfOperation.CyclicSyncVelocity);			
				CngToVelocityState := CngToVelocityState +1;
			END_IF
		END_IF	
	
	5:	
		DelayBeforeChangimeMode.IN := TRUE;
		DelayBeforeChangimeMode.PT := T#10S;
		IF DelayBeforeChangimeMode.Q THEN
			rAxisBasicFB.AxisCtrlPtr^.Input.Command.Power := TRUE;
			IF rAxisBasicFB.AxisCtrlPtr^.Output.Status.AxisStatus.StandStill THEN
				CngToVelocityState := CngToVelocityState +1;
			END_IF
		END_IF	
	6:
		IF  rAxisBasicFB.Meth_WriteObj(TRUE, enumMotionObject.ACC_CLOSE_POS_ERR ,   rVelocityCtrl.Input.Parameter.CyclicVelocity    , Error =>Error ) THEN
			rAxisBasicFB.Meth_WriteObj(FALSE, enumMotionObject.ACC_CLOSE_POS_ERR ,0 );
			CngToVelocityState := CngToVelocityState +1;
		END_IF	
	
	7:	
		METH_ChangeToVelMode := TRUE;
END_CASE

DelayBeforeChangimeMode();

	IF CngToVelocityState <> PrevCngToVelocityState THEN
		
		fnLogMsg(ADR(LogMsg_0),LOG_INFO,'CngToVelocityState CurSt=%d LstSt=%d',CngToVelocityState,PrevCngToVelocityState,0);
		PrevCngToVelocityState := CngToVelocityState ;
	END_IF
END_METHOD

METHOD Meth_ExitVelCtrl : BOOL
VAR_INPUT
	Execute   : BOOL;
END_VAR

VAR_INST
	// Service Functions Variablea
	StopTrigger : Trigger ;
	ExitState  		 : SINT;
	PrevExitState   : SINT;
END_VAR

VAR_OUTPUT
	Error : BOOL;
END_VAR

IF StopTrigger.EDGEPOS(Execute) THEN
	ExitState  := 1;
	Meth_ExitVelCtrl := FALSE;
 	Meth_ReturnOrgPosCtrlValues(FALSE) ;
	Error := FALSE;
END_IF


IF StopTrigger.EDGENEG(Execute) THEN
	 PrevExitState := 0;
	 ExitState:= 0;
END_IF


CASE ExitState OF
	 		
	
	1:	 
		
//			
 //  	
		Delay(IN:=	FALSE);
		IF rAxisBasicFB.AxisCtrlPtr^.Output.Status.AxisStatus.StandStill = FALSE  AND rAxisBasicFB.AxisCtrlPtr^.Output.Status.AxisStatus.Disabled = FALSE THEN
		//	rAxisBasicFB.AxisCtrlPtr^.Input.Command.MoveVelocity := TRUE;	
		//	rAxisBasicFB.AxisCtrlPtr^.Input.Parameter.Velocity   := 100;
			rAxisBasicFB.AxisCtrlPtr^.Input.Command.Stop := TRUE;		
			ExitState := ExitState +1;
		ELSE
			ExitState := 3;
		END_IF	
					
   						
		
		
		
	2:
			IF (rAxisBasicFB.AxisCtrlPtr^.Output.Status.AxisStatus.StandStill OR rAxisBasicFB.AxisCtrlPtr^.Output.Status.AxisStatus.Disabled)				
			//IF rAxisBasicFB.AxisCtrlPtr^.Output.Status.MC_MoveVelocity.In_Velocity 
				 THEN
				Delay.PT := T#2S;
				Delay(IN:=	TRUE);
				IF Delay.Q THEN
					ExitState := ExitState +1;
				END_IF								
			END_IF

	
	3:
			rAxisBasicFB.AxisCtrlPtr^.Input.Command.Power := FALSE;

			ExitState := ExitState +1;

	4:
		IF rAxisBasicFB.AxisCtrlPtr^.Output.Status.AxisStatus.Disabled THEN
			IF ReadPosCtrlParamDone THEN
				IF  rAxisBasicFB.Meth_WriteObj(TRUE, enumMotionObject.ACC_CLOSE_POS_ERR ,  rVelocityCtrl.Output.monitor.OrgAccToCloseThePosError, Error =>Error ) THEN
					rAxisBasicFB.Meth_WriteObj(FALSE, enumMotionObject.ACC_CLOSE_POS_ERR ,0 );
					ExitState := ExitState +1;
				END_IF
			ELSE	
				ExitState := ExitState +1;
			END_IF
			
		END_IF	
	

	5:
		IF ReadPosCtrlParamDone THEN
			IF Meth_ReturnOrgPosCtrlValues(TRUE) THEN
				ExitState := ExitState +1;
			END_IF
		ELSE	
			ExitState := ExitState +1;
		END_IF
	
	
	6:		
		IF rAxisBasicFB.Meth_WriteObj (TRUE, enumMotionobject.OPERATION_MODE,TO_LREAL(eDriveModeOfOperation.CyclicSyncMode)) THEN
			rAxisBasicFB.Meth_WriteObj (FALSE, enumMotionobject.OPERATION_MODE,0);
			Delay.IN := FALSE;
			ExitState := ExitState +1;
		END_IF
	7:
			Delay.IN := TRUE;
			Delay.PT := T#2S;
			Delay();
			IF Delay.Q THEN
				ExitState := ExitState +1;
				Delay.IN := FALSE;
			END_IF

	8:
 		Meth_ExitVelCtrl := TRUE;
		

	

END_CASE

	IF ExitState <> PrevExitState THEN
		
		fnLogMsg(ADR(LogMsg_0),LOG_INFO,'Exit Vel Ctrl CurSt=%d LstSt=%d',ExitState,PrevExitState,0);
		PrevExitState := ExitState ;
	END_IF
END_METHOD

METHOD Meth_InitSctrl : BOOL
VAR_INPUT
	Execute : BOOL;
END_VAR


VAR_OUTPUT
	Error : BOOL;
END_VAR
IF InitSctrlTrigger.EDGEPOS(Execute) THEN
	InitSctrlState  := 1;
	Meth_InitSctrl := FALSE;
	rAxisBasicFB.Meth_InitVelKP (FALSE,0);
	rAxisBasicFB.Meth_InitVelKI(FALSE,0);
	Error := FALSE;
END_IF


IF InitSctrlTrigger.EDGENEG(Execute) THEN
	
	 InitSctrlState:= 0;
END_IF


CASE InitSctrlState OF
	 
		
	1:
		 			
			IF rAxisBasicFB.Meth_InitVelKP (TRUE,(rVelocityCtrl.Input.Parameter.SctrlKp), Error=>Error) THEN
				OldSctrlKp := rVelocityCtrl.Input.Parameter.SctrlKp;
				InitSctrlState := InitSctrlState +1;
				rAxisBasicFB.Meth_InitVelKP (FALSE,rVelocityCtrl.Input.Parameter.SctrlKp);
			END_IF	
  
			

	2:
	
		IF rAxisBasicFB.Meth_InitVelKI(TRUE,(rVelocityCtrl.Input.Parameter.SctrlKi), Error=>Error) THEN
			rAxisBasicFB.Meth_InitVelKP (FALSE,rVelocityCtrl.Input.Parameter.SctrlKi);
			OldSctrlKi := rVelocityCtrl.Input.Parameter.SctrlKi ;
			InitSctrlState := InitSctrlState +1;
		END_IF	

		IF Error THEN
		//	
		END_IF
		
	3:		
		rAxisBasicFB.Meth_WriteObj(FALSE,enumMotionObject.VEL_KI,0);
		rVelocityCtrl.Output.Status.SctrlInitialized := TRUE;
		Meth_InitSctrl := TRUE; 
	END_CASE
END_METHOD

METHOD Meth_MoveVel : BOOL
VAR_INPUT
END_VAR
	rAxisBasicFB.AxisCtrlPtr^.Input.Parameter.Velocity 	   := rVelocityCtrl.Input.Parameter.CyclicVelocity;
	rAxisBasicFB.AxisCtrlPtr^.Input.Parameter.Acceleration := rVelocityCtrl.Input.Parameter.Acceleration;
	rAxisBasicFB.AxisCtrlPtr^.Input.Parameter.Deceleration := rVelocityCtrl.Input.Parameter.Deceleration;
	
	rAxisBasicFB.AxisCtrlPtr^.Input.Command.MoveVelocity := TRUE;
END_METHOD

METHOD Meth_ReadPosCtrlValues : BOOL
VAR_INPUT
	Execute : BOOL;
END_VAR


VAR_INST
	// Service Functions Variablea
		 
	ReadOrginalValuesTrigger : Trigger ;
	ReadOrginalValuesState   : SINT;
END_VAR	

VAR_OUTPUT
	Error : BOOL;	
END_VAR
IF ReadOrginalValuesTrigger.EDGEPOS(Execute) THEN
	ReadOrginalValuesState  := 1;
	Meth_ReadPosCtrlValues := FALSE;
	Error := FALSE;
	rAxisBasicFB.Meth_ReadObj(FALSE, enumMotionObject.MAX_TORQUE, Value =>rVelocityCtrl.Output.monitor.OrgMaxTorque, Error =>Error );
END_IF


IF ReadOrginalValuesTrigger.EDGENEG(Execute) THEN
	 rAxisBasicFB.Meth_ReadObj(FALSE, enumMotionObject.MAX_TORQUE, Value =>rVelocityCtrl.Output.monitor.OrgMaxTorque, Error =>Error );
	 ReadOrginalValuesState:= 0;
END_IF


CASE ReadOrginalValuesState OF
	 
		
	1:
		IF  rAxisBasicFB.Meth_ReadObj(TRUE, enumMotionObject.TORQUE_OFFSET, Value =>rVelocityCtrl.Output.monitor.OrgCyclicTorque, Error =>Error ) THEN
			fnLogMsg(ADR(LogMsg_0),LOG_INFO,'TORQUE_OFFSET org=%d',TO_DINT(rVelocityCtrl.Output.monitor.OrgCyclicTorque),0,0);
			rAxisBasicFB.Meth_ReadObj(FALSE, enumMotionObject.TORQUE_OFFSET  );
 			ReadOrginalValuesState := ReadOrginalValuesState +1;
			Error := FALSE;						
		END_IF
		IF Error THEN
			ReadOrginalValuesState := 33;
		END_IF
			
	2:
		IF  rAxisBasicFB.Meth_ReadObj(TRUE, enumMotionObject.VEL_KP, Value =>rVelocityCtrl.Output.monitor.OrgSctrlKp, Error =>Error ) THEN
			rVelocityCtrl.Output.monitor.OrgVelKp := rVelocityCtrl.Output.monitor.OrgSctrlKp;
			
			fnLogMsg(ADR(LogMsg_0),LOG_INFO,'VEL_KP org=%d',TO_DINT(rVelocityCtrl.Output.monitor.OrgSctrlKp),0,0);
			rAxisBasicFB.Meth_ReadObj(FALSE, enumMotionObject.TORQUE_OFFSET  );
 			ReadOrginalValuesState := ReadOrginalValuesState +1;
		END_IF
	3:
		IF  rAxisBasicFB.Meth_ReadObj(TRUE, enumMotionObject.VEL_KI, Value =>rVelocityCtrl.Output.monitor.OrgSctrlKi, Error =>Error ) THEN
			fnLogMsg(ADR(LogMsg_0),LOG_INFO,'VEL_KI org=%d',TO_DINT(rVelocityCtrl.Output.monitor.OrgSctrlKi),0,0);
			rAxisBasicFB.Meth_ReadObj(FALSE, enumMotionObject.TORQUE_OFFSET  );
 			ReadOrginalValuesState := ReadOrginalValuesState +1;
		END_IF
	
	4:
		IF rAxisBasicFB.Meth_ReadObj (TRUE, enumMotionobject.GAIN_SCHEDULE, Value =>rVelocityCtrl.Output.monitor.OrgGainCtrl, Error =>Error) THEN
				fnLogMsg(ADR(LogMsg_0),LOG_INFO,'GAIN_SCHEDULE org=%d',TO_DINT(rVelocityCtrl.Output.monitor.OrgGainCtrl),0,0);			
				rAxisBasicFB.Meth_ReadObj(FALSE, enumMotionObject.TORQUE_OFFSET  );
				ReadOrginalValuesState := ReadOrginalValuesState +1;						
		END_IF		
		
	5:
	

			IF rAxisBasicFB.Meth_ReadObj (TRUE, enumMotionobject.ACC_CLOSE_POS_ERR, Value =>rVelocityCtrl.Output.monitor.OrgAccToCloseThePosError, Error =>Error) THEN
				fnLogMsg(ADR(LogMsg_0),LOG_INFO,'ACC_CLOSE_POS_ERR org=%d',TO_DINT(rVelocityCtrl.Output.monitor.OrgAccToCloseThePosError),0,0);			
				rAxisBasicFB.Meth_ReadObj(FALSE, enumMotionObject.TORQUE_OFFSET  );
				ReadOrginalValuesState := ReadOrginalValuesState +1;						
			END_IF		

	7:		
		ReadPosCtrlParamDone := TRUE;
		Meth_ReadPosCtrlValues := TRUE; 
	END_CASE
END_METHOD

METHOD Meth_ReturnOrgPosCtrlValues : BOOL
VAR_INPUT
	Execute : BOOL;
END_VAR


VAR_INST
	// Service Functions Variablea
	ReturnOrginalTrigger : Trigger ;
	ReturnOrginalState   : SINT;
END_VAR	

VAR_OUTPUT
	Error : BOOL;
END_VAR
IF ReturnOrginalTrigger.EDGEPOS(Execute) THEN
	ReturnOrginalState  := 1;
	Meth_ReturnOrgPosCtrlValues := FALSE;
	Error := FALSE;
	rAxisBasicFB.Meth_WriteObj(FALSE, enumMotionObject.MAX_TORQUE, rVelocityCtrl.Output.monitor.OrgMaxTorque, Error =>Error );
	fnLogMsg(ADR(LogMsg_0),LOG_INFO,'VelCtrl Start Return Org Values',0,0,0);
END_IF


IF ReturnOrginalTrigger.EDGENEG(Execute) THEN
	 rAxisBasicFB.Meth_WriteObj(FALSE, enumMotionObject.MAX_TORQUE,  rVelocityCtrl.Output.monitor.OrgMaxTorque, Error =>Error );
	 ReturnOrginalState:= 0;
END_IF


CASE ReturnOrginalState OF
	 
		
	1:	
		IF  rAxisBasicFB.Meth_WriteObj(TRUE, enumMotionObject.GAIN_SCHEDULE,  rVelocityCtrl.Output.monitor.OrgGainCtrl, Error =>Error ) THEN
			rAxisBasicFB.Meth_WriteObj(FALSE, enumMotionObject.GAIN_SCHEDULE ,0 );
 			ReturnOrginalState := ReturnOrginalState +1;
		END_IF		
			
	2:
		IF  rAxisBasicFB.Meth_WriteObj(TRUE, enumMotionObject.VEL_KP,  rVelocityCtrl.Output.monitor.OrgSctrlKp, Error =>Error ) THEN
			rAxisBasicFB.Meth_WriteObj(FALSE,enumMotionObject.VEL_KP,0  );
 			ReturnOrginalState := ReturnOrginalState +1;
		END_IF
	3:
		IF  rAxisBasicFB.Meth_WriteObj(TRUE, enumMotionObject.VEL_KI,  rVelocityCtrl.Output.monitor.OrgSctrlKi, Error =>Error ) THEN
			rAxisBasicFB.Meth_WriteObj(FALSE, enumMotionObject.VEL_KP ,0 );
 			ReturnOrginalState := ReturnOrginalState +1;
		END_IF
	
	4:
		IF  rAxisBasicFB.Meth_WriteObj(TRUE, enumMotionObject.TORQUE_OFFSET, rVelocityCtrl.Output.monitor.OrgCyclicTorque , Error =>Error ) THEN
			rAxisBasicFB.Meth_WriteObj(FALSE, enumMotionObject.VEL_KP ,0 );
 			ReturnOrginalState := ReturnOrginalState +1;
		END_IF
		
	5:
	
	        IF rAxisBasicFB.Meth_WriteObj(TRUE, enumMotionObject.MAX_TORQUE,rVelocityCtrl.Output.monitor.OrgMaxTorque   , Error =>Error ) THEN	
				rAxisBasicFB.Meth_WriteObj(FALSE, enumMotionObject.VEL_KP ,0 );									
				rAxisBasicFB.Meth_WriteObj(FALSE, enumMotionObject.VEL_KP ,0 );
				ReturnOrginalState := ReturnOrginalState +1;					
			END_IF	
	
	6:			
		fnLogMsg(ADR(LogMsg_0),LOG_INFO,'VelCtrl Return Org Values Done',0,0,0);
		Meth_ReturnOrgPosCtrlValues := TRUE; 
	END_CASE
END_METHOD

METHOD Meth_Stop : BOOL
VAR_INPUT
	Execute   : BOOL;
END_VAR

VAR_INST
	// Service Functions Variablea
	StopTrigger : Trigger ;
	StopState   : SINT;
	
END_VAR

VAR_OUTPUT
	Error : BOOL;
END_VAR

IF StopTrigger.EDGEPOS(Execute) THEN
	StopState  := 1;
	Meth_Stop := FALSE;
 	Meth_ReturnOrgPosCtrlValues(FALSE) ;
	Error := FALSE;
END_IF


IF StopTrigger.EDGENEG(Execute) THEN
	
	 StopState:= 0;
END_IF


CASE StopState OF
 		
	
	1:	 
		
		rAxisBasicFB.AxisCtrlPtr^.Input.Command.Stop := TRUE;			
   		StopState := StopState +1;				
		Delay(IN:=	FALSE);
		
	2:
			IF rAxisBasicFB.AxisCtrlPtr^.Output.Status.AxisStatus.StandStill OR rAxisBasicFB.AxisCtrlPtr^.Output.Status.AxisStatus.Disabled THEN
				StopState := StopState +1;								
			END_IF

	


	3:
 		Meth_Stop := TRUE;
		

	

END_CASE
END_METHOD

METHOD PRIVATE ResetAll_MC_FB : BOOL
VAR_INPUT
END_VAR

		ResetAll_MC_FB := FALSE ;
				

		{warning disable C0371}
		//Warning: Access to VAR_IN_OUT <Var> declared in <POU> from external context <Method/Transition/Property>

		{warning restore C0371}
		
		
		memset(ADR(rVelocityCtrl.Input.Command) ,0 ,SIZEOF(rVelocityCtrl.Input.Command));
		memset(ADR(rVelocityCtrl.Output.Status) ,0 ,SIZEOF(rVelocityCtrl.Output.Status));
		
		ResetAll_MC_FB := TRUE ;
END_METHOD

END_FUNCTION_BLOCK

// ---- POUs/Lib/Motion/CanOpenAxis/Lti/LtiBasicAxis_FB.TcPOU
FUNCTION_BLOCK PUBLIC LtiBasicAxis_FB EXTENDS CoE_BasicAxis_FB  
VAR_INPUT		
	pDigIn: 	POINTER TO DINT;
END_VAR
VAR_IN_OUT	
END_VAR
VAR_OUTPUT	
END_VAR

VAR
	
	
END_VAR



SUPER^(AxisRef:=AxisRef);

METHOD GetErrCanAdr : BOOL
VAR_INPUT
END_VAR


VAR
		
END_VAR
SUPER^.GetCanOpenAdr();		
CoeErrIdIndex	 := 16#2027;
CoeErrIdSubIndex := 0;
END_METHOD

METHOD ReadActualTorque : LREAL
VAR_INPUT
END_VAR
VAR_INST
	
	
	
END_VAR

IF THIS^.TorqueReadEnable THEN			
	tmp_ActualTorque:= io_ActualTorqueReal;		
END_IF

ReadActualTorque:= tmp_ActualTorque;
END_METHOD

METHOD ReadDriveError
VAR_INPUT
END_VAR
VAR_INST 
	ErrIdIndex	: WORD;
END_VAR
DriveError := AxisRef.NcToPlc.StateDWord AND 16#10000000 ;
ErrIdIndex	:= 16#2027; // decimal = 39;
END_METHOD

END_FUNCTION_BLOCK

// ---- POUs/Lib/Motion/CanOpenAxis/Nidic/NidicBasicAxis_FB.TcPOU
FUNCTION_BLOCK PUBLIC NidicBasicAxis_FB EXTENDS CoE_BasicAxis_FB  
VAR_INPUT		
		
END_VAR
VAR_IN_OUT	
END_VAR
VAR_OUTPUT	
END_VAR

VAR
	DebugError					: UINT;
	
END_VAR


AxisCtrlPtr^.Input.Parameter.Drive.eDriveType := enumDriveType.eNidec;	
AxisCtrlPtr^.Input.Parameter.Drive.VendorNameID := eVendorNameID.Nidec;	
SUPER^(AxisRef:=AxisRef);

AxisCtrlPtr^.Output.Status.DriveEnable			:= io_StatusWord.0;	// DS-402 Status word bit 0 = Ready to switch on

METHOD CreateDriveErrMsgDetails : enumMotorEvents
VAR_INPUT
	ErrorId			: UDINT;
END_VAR

CASE ErrorId OF
	
	16#0:
		CreateDriveErrMsgDetails := enumMotorEvents.NoEvents;
		fnLogMsg(ADR(LogMsg_0),LOG_ERROR,'Nidic Drive ErrorId %d  ,No error',UDINT_TO_DINT(ErrorId),0,0);
	16#FF01: 
		CreateDriveErrMsgDetails := enumMotorEvents.MotorGeneralError ;
		fnLogMsg(ADR(LogMsg_0),LOG_ERROR,'Nidic Drive ErrorId %d Generic Error',UDINT_TO_DINT(ErrorId),0,0);
	16#2300:
		CreateDriveErrMsgDetails := enumMotorEvents.MotorSupplyError ;
		fnLogMsg(ADR(LogMsg_0),LOG_ERROR,'Nidic Drive ErrorId %d Current, device outputside',UDINT_TO_DINT(ErrorId),0,0);	
	16#3130:
		CreateDriveErrMsgDetails := enumMotorEvents.MotorSupplyError ;
		fnLogMsg(ADR(LogMsg_0),LOG_ERROR,'Nidic Drive ErrorId %d Phase failure',UDINT_TO_DINT(ErrorId),0,0);	
	
	16#2230:
		CreateDriveErrMsgDetails := enumMotorEvents.MotorSupplyError ;
		fnLogMsg(ADR(LogMsg_0),LOG_ERROR,'Nidic Drive ErrorId %d Short circuit/ground leakage',UDINT_TO_DINT(ErrorId),0,0);	

	16#3210:
		CreateDriveErrMsgDetails := enumMotorEvents.MotorSupplyError ;
		fnLogMsg(ADR(LogMsg_0),LOG_ERROR,'Nidic Drive ErrorId %d DC link over-voltage',UDINT_TO_DINT(ErrorId),0,0);	

		 
	16#3230:
		CreateDriveErrMsgDetails := enumMotorEvents.MotorStalled; 
		fnLogMsg(ADR(LogMsg_0),LOG_ERROR,'Nidic Drive ErrorId %d Load error, Low Load',UDINT_TO_DINT(ErrorId),0,0);
	16#4310:
		CreateDriveErrMsgDetails := enumMotorEvents.MotorOverTemp; 
		fnLogMsg(ADR(LogMsg_0),LOG_ERROR,'Nidic Drive ErrorId %d Excess temperature drive',UDINT_TO_DINT(ErrorId),0,0);
	16#5112:
		 CreateDriveErrMsgDetails := enumMotorEvents.MotorSupplyError;
		 fnLogMsg(ADR(LogMsg_0),LOG_ERROR,'Nidic Drive ErrorId %d Supply low voltage' ,UDINT_TO_DINT(ErrorId),0,0);

	16#5200:
		 CreateDriveErrMsgDetails := enumMotorEvents.MotorGeneralError;
		 fnLogMsg(ADR(LogMsg_0),LOG_ERROR,'Nidic Drive ErrorId %d Control device hardware',UDINT_TO_DINT(ErrorId),0,0);

	16#5400:
		CreateDriveErrMsgDetails := enumMotorEvents.MotorSupplyError; 
		fnLogMsg(ADR(LogMsg_0),LOG_ERROR,'Nidic Drive ErrorId %d Power section',UDINT_TO_DINT(ErrorId),0,0);

	16#5510:
		CreateDriveErrMsgDetails := enumMotorEvents.MotorGeneralError; 
		fnLogMsg(ADR(LogMsg_0),LOG_ERROR, 'Nidic Drive ErrorId %d RAM Allocation',UDINT_TO_DINT(ErrorId),0,0);
	16#5530:
		CreateDriveErrMsgDetails := enumMotorEvents.MotorGeneralError; 
		fnLogMsg(ADR(LogMsg_0),LOG_ERROR, 'Nidic Drive ErrorId %d Data storage (Non-volatile)',UDINT_TO_DINT(ErrorId),0,0);

	16#5430:
		CreateDriveErrMsgDetails := enumMotorEvents.MotorSupplyError; 
		fnLogMsg(ADR(LogMsg_0),LOG_ERROR,'Nidic Drive ErrorId %d  Input stages 94 - Rectifier set up',UDINT_TO_DINT(ErrorId),0,0);
	16#5440:
		CreateDriveErrMsgDetails := enumMotorEvents.MotorSupplyError; 
		fnLogMsg(ADR(LogMsg_0),LOG_ERROR, 'Nidic Drive ErrorId %d Contacts 226 - Soft Start',UDINT_TO_DINT(ErrorId),0,0);
	16#6010:
		CreateDriveErrMsgDetails := enumMotorEvents.MotorGeneralError;
 		fnLogMsg(ADR(LogMsg_0),LOG_ERROR, 'Nidic Drive ErrorId %d Software reset',UDINT_TO_DINT(ErrorId),0,0);

	16#6320:
		CreateDriveErrMsgDetails := enumMotorEvents.PLCIllegalParam; 
		fnLogMsg(ADR(LogMsg_0),LOG_ERROR,'Nidic Drive ErrorId %d Parameter Error',UDINT_TO_DINT(ErrorId),0,0);

	16#7112:
		CreateDriveErrMsgDetails := enumMotorEvents.BreakResistorError; 
		fnLogMsg(ADR(LogMsg_0),LOG_ERROR, 'Nidic Drive ErrorId %d Brake chopper over',UDINT_TO_DINT(ErrorId),0,0);//????

	16#7113:
		CreateDriveErrMsgDetails := enumMotorEvents.MotorSupplyError; 
		fnLogMsg(ADR(LogMsg_0),LOG_ERROR,'Nidic Drive ErrorId %d  Protective circuit break',UDINT_TO_DINT(ErrorId),0,0);
(*chopper 10 - Th Brake Res*)
	16#7120: 
		CreateDriveErrMsgDetails := enumMotorEvents.DriveNotReady;
		fnLogMsg(ADR(LogMsg_0),LOG_ERROR,'Nidic Drive ErrorId %d  Motor Autotune',UDINT_TO_DINT(ErrorId),0,0);

	16#7122:
		CreateDriveErrMsgDetails := enumMotorEvents.DriveComError; 
		fnLogMsg(ADR(LogMsg_0),LOG_ERROR,'Nidic Drive ErrorId %d  Motor error OR commutation malfunction',UDINT_TO_DINT(ErrorId),0,0);
	16#7300:
		CreateDriveErrMsgDetails := enumMotorEvents.MotorFeedBackErr; 
		fnLogMsg(ADR(LogMsg_0),LOG_ERROR, 'Nidic Drive ErrorId %d Sensor Error',UDINT_TO_DINT(ErrorId),0,0);

	16#7310:
		CreateDriveErrMsgDetails := enumMotorEvents.MotorSpeedError; 
		fnLogMsg(ADR(LogMsg_0),LOG_ERROR,'Nidic Drive ErrorId %d  Speed 7 - Over speed',UDINT_TO_DINT(ErrorId),0,0);
	16#7500:
		CreateDriveErrMsgDetails := enumMotorEvents.DriveComError; 
		fnLogMsg(ADR(LogMsg_0),LOG_ERROR,'Nidic Drive ErrorId %d Communication 90 - Power Comms',UDINT_TO_DINT(ErrorId),0,0);
(*103 - Interconnect*)
	16#7600:
		CreateDriveErrMsgDetails := enumMotorEvents.MotorGeneralError; 
		fnLogMsg(ADR(LogMsg_0),LOG_ERROR,'Nidic Drive ErrorId %d Data storage (external)',UDINT_TO_DINT(ErrorId),0,0);	
		
		
	ELSE
		fnLogMsg(ADR(LogMsg_0),LOG_ERROR,'unknown Nidic Drive ErrorId %d ',UDINT_TO_DINT(ErrorId),0,0);
		CreateDriveErrMsgDetails := enumMotorEvents.NoEvents;
	END_CASE
END_METHOD

METHOD  INIT_Specific : BOOL 
VAR_INPUT
	bStart: 					BOOL;
END_VAR
VAR_INST	
	ComDelay:	TON;
	Nidec_Init_State : INT ;
	ExecuteTrig: 	Trigger;
END_VAR
IF ExecuteTrig.EDGEPOS(bStart) THEN
	INIT_Specific := FALSE ;
	IF AxisCtrlPtr^.Input.Parameter.Drive.bDisableFoE_Transfer THEN 
		Nidec_Init_State:= 5;//10;
	ELSE
		Nidec_Init_State:= 1;
	END_IF
END_IF


IF ExecuteTrig.EDGENEG(bStart) THEN
	Nidec_Init_State := 0;
END_IF	

	
CASE Nidec_Init_State OF							
						
	1:	
		Nidec_Init_State:= 5;			
	5:
		ReadInitDriveParID(FALSE);
		Nidec_Init_State:=	6;
		
	6:
		IF ReadInitDriveParID(TRUE) THEN
			Nidec_Init_State:=	10;
		END_IF
	
	
	10:
		
		Nidec_Init_State := 0 ;
		INIT_Specific := TRUE ;
		AxisCtrlPtr^.Output.Status.AxisInitDone := TRUE ;
		AxisCtrlPtr^.Output.Status.ReadyForCmd := TRUE ;
END_CASE
END_METHOD

METHOD ReadInitDriveParID : BOOL
VAR_INPUT
	bStart : BOOL;
END_VAR

VAR_INST
	ExecuteTrig_1: 		Trigger;
	State_InitSpecific_1: INT;
END_VAR

IF ExecuteTrig_1.EDGEPOS(bStart) THEN
	ReadInitDriveParID		:= FALSE;
	State_InitSpecific_1	:= 1;		
END_IF

IF ExecuteTrig_1.EDGENEG(bStart) THEN
	State_InitSpecific_1	:= 0;	
	ReadInitDriveParID		:= FALSE;
END_IF

CASE State_InitSpecific_1 OF

 
	
	1:
		SUPER^.EcCoeSdoRead(FALSE);
		CoeSdoRW.Input.Read.nIndex		:= DINT_TO_WORD(eNidecDriveParID.Menue05);
		CoeSdoRW.Input.Read.nSubIndex	:= 7;
		CoeSdoRW.Input.Read.pDstBuf		:= ADR(CoeRead_RatedCurrent);
		CoeSdoRW.Input.Read.cbBufLen	:= SIZEOF(CoeRead_RatedCurrent);
		State_InitSpecific_1	:= 2;
		
	2:
		IF SUPER^.EcCoeSdoRead(TRUE) THEN	
			State_InitSpecific_1	:= 3;
		END_IF
		
	3:
		SUPER^.EcCoeSdoRead(FALSE);
		CoeSdoRW.Input.Read.nIndex		:= DINT_TO_WORD(eNidecDriveParID.Menue04);
		CoeSdoRW.Input.Read.nSubIndex	:= 41;
		CoeSdoRW.Input.Read.pDstBuf		:= ADR(CoeRead_RatedTorque);
		CoeSdoRW.Input.Read.cbBufLen	:= SIZEOF(CoeRead_RatedTorque);
		State_InitSpecific_1	:= 4;
		
	4:
		IF SUPER^.EcCoeSdoRead(TRUE) THEN
			AxisCtrlPtr^.Input.Parameter.RatedCurrent	:= UDINT_TO_LREAL(CoeRead_RatedCurrent) / 1000.0;
			AxisCtrlPtr^.Input.Parameter.Ratedtorque	:= UDINT_TO_LREAL(CoeRead_RatedTorque) / 100.0;
			ReadInitDriveParID		:= TRUE;	
			State_InitSpecific_1	:= 0;
		END_IF
		
		
 
		
END_CASE
END_METHOD

END_FUNCTION_BLOCK

// ---- POUs/Lib/Motion/CanOpenAxis/Nidic/NidicIntegratedAxis_FB.TcPOU
FUNCTION_BLOCK PUBLIC NidicIntegratedAxis_FB EXTENDS CoE_BasicAxis_FB  
VAR_INPUT		
		
END_VAR
VAR_IN_OUT	
END_VAR
VAR_OUTPUT	
END_VAR

VAR
	DebugError					: UINT;
	
END_VAR


AxisCtrlPtr^.Input.Parameter.Drive.eDriveType := enumDriveType.eIntegratedNidec;	
AxisCtrlPtr^.Input.Parameter.Drive.VendorNameID := eVendorNameID.Nidec;	
SUPER^(AxisRef:=AxisRef);

AxisCtrlPtr^.Output.Status.DriveEnable			:= io_StatusWord.4 AND  (io_StatusWord.0) ;	// DS-402 Status word bit 0 = Ready to switch on

METHOD CreateDriveErrMsgDetails : enumMotorEvents
VAR_INPUT
	ErrorId			: UDINT;
END_VAR

CASE ErrorId OF
	
	16#0:
		CreateDriveErrMsgDetails := enumMotorEvents.NoEvents;
		fnLogMsg(ADR(LogMsg_0),LOG_ERROR,'NidicInt Drive ErrorId %d  ,No error',UDINT_TO_DINT(ErrorId),0,0);
	16#2220:
		CreateDriveErrMsgDetails := enumMotorEvents.MotorSupplyError ;
		fnLogMsg(ADR(LogMsg_0),LOG_ERROR,'NidicInt Drive ErrorId %d Current, device outputside',UDINT_TO_DINT(ErrorId),0,0);	
	16#2250:
		CreateDriveErrMsgDetails := enumMotorEvents.MotorSupplyError ;
		fnLogMsg(ADR(LogMsg_0),LOG_ERROR,'NidicInt Drive ErrorId %d Short circuit/ground leakage',UDINT_TO_DINT(ErrorId),0,0);	

	16#2351:
		CreateDriveErrMsgDetails := enumMotorEvents.MotorSupplyError ;
		fnLogMsg(ADR(LogMsg_0),LOG_ERROR,'I2T THERMAL STATE LOAD EVEL WARNING',UDINT_TO_DINT(ErrorId),0,0);	
	
		
	16#3130:
		CreateDriveErrMsgDetails := enumMotorEvents.MotorSupplyError ;
		fnLogMsg(ADR(LogMsg_0),LOG_ERROR,'NidicInt Drive ErrorId %d Phase failure',UDINT_TO_DINT(ErrorId),0,0);
	
	16#3131:
		CreateDriveErrMsgDetails := enumMotorEvents.MotorSupplyError ;
		fnLogMsg(ADR(LogMsg_0),LOG_ERROR,'NidicInt Drive ErrorId %d Phase 1 failure',UDINT_TO_DINT(ErrorId),0,0);	

	16#3132:
		CreateDriveErrMsgDetails := enumMotorEvents.MotorSupplyError ;
		fnLogMsg(ADR(LogMsg_0),LOG_ERROR,'NidicInt Drive ErrorId %d Phase 2 failure',UDINT_TO_DINT(ErrorId),0,0);	
	
	16#3133:
		CreateDriveErrMsgDetails := enumMotorEvents.MotorSupplyError ;
		fnLogMsg(ADR(LogMsg_0),LOG_ERROR,'NidicInt Drive ErrorId %d Phase 3 failure',UDINT_TO_DINT(ErrorId),0,0);	
	

	16#3210:
		CreateDriveErrMsgDetails := enumMotorEvents.MotorSupplyError ;
		fnLogMsg(ADR(LogMsg_0),LOG_ERROR,'NidicInt Drive ErrorId %d DC link over-voltage',UDINT_TO_DINT(ErrorId),0,0);	

		 
	16#3220:
		CreateDriveErrMsgDetails := enumMotorEvents.MotorSupplyError; 
		fnLogMsg(ADR(LogMsg_0),LOG_ERROR,'NidicInt Drive ErrorId %d DC Link under voltage',UDINT_TO_DINT(ErrorId),0,0);
	
	16#3331:
		CreateDriveErrMsgDetails := enumMotorEvents.MotorSupplyError; 
		fnLogMsg(ADR(LogMsg_0),LOG_ERROR,'NidicInt Drive ErrorId %d FIELD CIRCUIT INTERRUPTED',UDINT_TO_DINT(ErrorId),0,0);
	
	
	16#4210:
		CreateDriveErrMsgDetails := enumMotorEvents.MotorOverTemp; 
		fnLogMsg(ADR(LogMsg_0),LOG_ERROR,'NidicInt Drive ErrorId %d Excess temperature drive',UDINT_TO_DINT(ErrorId),0,0);
		
	16#4310:
		CreateDriveErrMsgDetails := enumMotorEvents.MotorOverTemp; 
		fnLogMsg(ADR(LogMsg_0),LOG_ERROR,'NidicInt Drive ErrorId %d Excess temperature device',UDINT_TO_DINT(ErrorId),0,0);		
		

	16#5300:
		 CreateDriveErrMsgDetails := enumMotorEvents.MotorGeneralError;
		 fnLogMsg(ADR(LogMsg_0),LOG_ERROR,'NidicInt Drive ErrorId %d Control device hardware',UDINT_TO_DINT(ErrorId),0,0);

	16#6010:
		CreateDriveErrMsgDetails := enumMotorEvents.MotorGeneralError;
 		fnLogMsg(ADR(LogMsg_0),LOG_ERROR, 'NidicInt Drive ErrorId %d Software reset',UDINT_TO_DINT(ErrorId),0,0);

	16#6320:
		CreateDriveErrMsgDetails := enumMotorEvents.PLCIllegalParam; 
		fnLogMsg(ADR(LogMsg_0),LOG_ERROR,'NidicInt Drive ErrorId %d Parameter Error',UDINT_TO_DINT(ErrorId),0,0);


(*chopper 10 - Th Brake Res*)

	16#7121:
		CreateDriveErrMsgDetails := enumMotorEvents.MotorStalled; 
		fnLogMsg(ADR(LogMsg_0),LOG_ERROR,'NidicInt Drive ErrorId %d  Motor error OR commutation malfunction',UDINT_TO_DINT(ErrorId),0,0);
	16#7300:
		CreateDriveErrMsgDetails := enumMotorEvents.MotorFeedBackErr; 
		fnLogMsg(ADR(LogMsg_0),LOG_ERROR, 'NidicInt Drive ErrorId %d Sensor Error',UDINT_TO_DINT(ErrorId),0,0);

	16#7500:
		CreateDriveErrMsgDetails := enumMotorEvents.DriveComError; 
		fnLogMsg(ADR(LogMsg_0),LOG_ERROR,'NidicInt Drive ErrorId %d Communication 90 - Power Comms',UDINT_TO_DINT(ErrorId),0,0);

	
		
	ELSE
		fnLogMsg(ADR(LogMsg_0),LOG_ERROR,'unknown NidicInt Drive ErrorId %d ',UDINT_TO_DINT(ErrorId),0,0);
		CreateDriveErrMsgDetails := enumMotorEvents.NoEvents;
	END_CASE
END_METHOD

METHOD  INIT_Specific : BOOL 
VAR_INPUT
	bStart: 					BOOL;
END_VAR
VAR_INST	
	ComDelay:	TON;
	Nidec_Init_State : INT ;
	ExecuteTrig: 	Trigger;
END_VAR
IF ExecuteTrig.EDGEPOS(bStart) THEN
	INIT_Specific := FALSE ;
	IF AxisCtrlPtr^.Input.Parameter.Drive.bDisableFoE_Transfer THEN 
		Nidec_Init_State:= 5;//10;
	ELSE
		Nidec_Init_State:= 1;
	END_IF
END_IF


IF ExecuteTrig.EDGENEG(bStart) THEN
	Nidec_Init_State := 0;
END_IF	

	
CASE Nidec_Init_State OF							
						
	1:	
		Nidec_Init_State:= 5;			
	5:
		ReadInitDriveParID(FALSE);
		Nidec_Init_State:=	6;
		
	6:
		IF ReadInitDriveParID(TRUE) THEN
			Nidec_Init_State:=	10;
		END_IF
	
	
	10:
		
		Nidec_Init_State := 0 ;
		INIT_Specific := TRUE ;
		AxisCtrlPtr^.Output.Status.AxisInitDone := TRUE ;
		AxisCtrlPtr^.Output.Status.ReadyForCmd := TRUE ;
END_CASE
END_METHOD

METHOD ReadInitDriveParID : BOOL
VAR_INPUT
	bStart : BOOL;
END_VAR

VAR_INST
	ExecuteTrig_1: 		Trigger;
	State_InitSpecific_1: INT;
END_VAR

IF ExecuteTrig_1.EDGEPOS(bStart) THEN
	ReadInitDriveParID		:= FALSE;
	State_InitSpecific_1	:= 1;		
END_IF

IF ExecuteTrig_1.EDGENEG(bStart) THEN
	State_InitSpecific_1	:= 0;	
	ReadInitDriveParID		:= FALSE;
END_IF

CASE State_InitSpecific_1 OF

	0:
	
	1:
		SUPER^.EcCoeSdoRead(FALSE);
		CoeSdoRW.Input.Read.nIndex		:= DINT_TO_WORD(eNidecDriveParID.Menue05);
		CoeSdoRW.Input.Read.nSubIndex	:= 7;
		CoeSdoRW.Input.Read.pDstBuf		:= ADR(CoeRead_RatedCurrent);
		CoeSdoRW.Input.Read.cbBufLen	:= SIZEOF(CoeRead_RatedCurrent);
		State_InitSpecific_1	:= 2;
		
	2:
		IF SUPER^.EcCoeSdoRead(TRUE) THEN	
			State_InitSpecific_1	:= 3;
		END_IF
		
	3:
		SUPER^.EcCoeSdoRead(FALSE);
		CoeSdoRW.Input.Read.nIndex		:= DINT_TO_WORD(eNidecDriveParID.Menue04);
		CoeSdoRW.Input.Read.nSubIndex	:= 41;
		CoeSdoRW.Input.Read.pDstBuf		:= ADR(CoeRead_RatedTorque);
		CoeSdoRW.Input.Read.cbBufLen	:= SIZEOF(CoeRead_RatedTorque);
		State_InitSpecific_1	:= 4;
		
	4:
		IF SUPER^.EcCoeSdoRead(TRUE) THEN
			AxisCtrlPtr^.Input.Parameter.RatedCurrent	:= UDINT_TO_LREAL(CoeRead_RatedCurrent) / 1000.0;
			AxisCtrlPtr^.Input.Parameter.Ratedtorque	:= UDINT_TO_LREAL(CoeRead_RatedTorque) / 100.0;
			ReadInitDriveParID		:= TRUE;	
			State_InitSpecific_1	:= 0;
		END_IF
		
		
 
		
END_CASE
END_METHOD

END_FUNCTION_BLOCK

// ---- POUs/Lib/Motion/CanOpenAxis/ServTronix/ServoTronixBasicAxis_FB.TcPOU
FUNCTION_BLOCK PUBLIC ServoTronixBasicAxis_FB EXTENDS CoE_BasicAxis_FB  
VAR_INPUT		
	
END_VAR
VAR_IN_OUT	
END_VAR
VAR_OUTPUT	
END_VAR

VAR
	
	
END_VAR



SUPER^(AxisRef:=AxisRef);

METHOD ReadActualTorque : LREAL
VAR_INPUT
END_VAR
VAR_INST
	
END_VAR
CASE ReadTorqueState OF 
	
	0: 
		IF THIS^.TorqueReadEnable THEN			
			ReadTorqueState	:= 5;			
		END_IF
						
	5:
		IF AxisRef.Status.Operational THEN
			
			FB_EcCoeSdoRead_RatedTorque(
						sNetId		:= AxisCtrlPtr^.Input.Parameter.ecNetId ,
						nSlaveAddr	:= ULINT_TO_UINT(AxisCtrlPtr^.Input.Parameter.Drive.EtherCatAddr.Value) , 
						nSubIndex	:=, 
						nIndex		:= 16#6076 , 
						pDstBuf		:= ADR(CoeRead_RatedTorque), 
						cbBufLen	:= SIZEOF(CoeRead_RatedTorque), 
						bExecute	:= FALSE, 
						tTimeout	:= T#10S, 
						bBusy		=> , 
						bError		=> , 
						nErrId		=> 
						);
			ReadTorqueState	:= 10;
		END_IF	
	10: // Can Over Ethercat
		FB_EcCoeSdoRead_RatedTorque.bExecute	:= TRUE;
		
		ReadTorqueState	:= 20;
	20:
		IF FB_EcCoeSdoRead_RatedTorque.bError = TRUE THEN
			FB_EcCoeSdoRead_RatedTorque.bExecute	:= FALSE;
			ReadTorqueState	:= 5;
		ELSIF FB_EcCoeSdoRead_RatedTorque.bBusy = FALSE THEN
			FB_EcCoeSdoRead_RatedTorque.bExecute	:= FALSE;
			ReadTorqueState	:= 30;
		END_IF
		
	30:
		tmp_ActualTorque	:= TorqueConstant * (INT_TO_LREAL(THIS^.io_ActualTorque) / 1000.0) * 3.11;	
			
			
END_CASE

FB_EcCoeSdoRead_RatedTorque();
ReadActualTorque	:= tmp_ActualTorque;
END_METHOD

END_FUNCTION_BLOCK

// ---- POUs/Lib/Motion/CanOpenAxis/stepIM/stepIMBasicAxis_FB.TcPOU
FUNCTION_BLOCK PUBLIC stepIMBasicAxis_FB EXTENDS CoE_BasicAxis_FB  
VAR_INPUT		
	DigIn 		AT %I* : UDINT;
END_VAR
VAR_IN_OUT	
END_VAR


VAR

END_VAR


AxisCtrlPtr^.Input.Parameter.Drive.eDriveType := enumDriveType.stepIM;	
AxisCtrlPtr^.Input.Parameter.Drive.VendorNameID := eVendorNameID.Servotronics;
SUPER^(AxisRef:=AxisRef);

IF io_StatusWord<> 0 THEN
	AxisCtrlPtr^.Output.Status.DriveEnable := io_StatusWord.4;
ELSE	
	// Simulator 
	AxisCtrlPtr^.Output.Status.DriveEnable := TRUE;
END_IF	
 


//fbElmoIOsHandle(DigIn:=	pDigIn^);
//AxisCtrlPtr^.Output.Status.DriveEnable:=	fbElmoIOsHandle.bEnable;

METHOD CreateDriveErrMsgDetails : enumMotorEvents
VAR_INPUT
	ErrorId			: UDINT;
END_VAR
CASE ErrorId OF
	
	16#2214:
		CreateDriveErrMsgDetails := enumMotorEvents.MotorOverCurrent;
		fnLogMsg(ADR(LogMsg_0),LOG_ERROR,'StepIM Drive ErrorId %d  ,Over Current',UDINT_TO_DINT(ErrorId),0,0);
	16#2310: 
		CreateDriveErrMsgDetails := enumMotorEvents.PLCIllegalParam;
		fnLogMsg(ADR(LogMsg_0),LOG_ERROR,'StepIM Drive ErrorId %d Under Voltage',UDINT_TO_DINT(ErrorId),0,0);
	16#3110:
		CreateDriveErrMsgDetails := enumMotorEvents.MotorSupplyError;
		fnLogMsg(ADR(LogMsg_0),LOG_ERROR,'StepIM Drive ErrorId %d Over-voltage',UDINT_TO_DINT(ErrorId),0,0);
	16#3120:
		CreateDriveErrMsgDetails := enumMotorEvents.MotorSupplyError ;
		fnLogMsg(ADR(LogMsg_0),LOG_ERROR,'StepIM Drive ErrorId %d Under-voltage',UDINT_TO_DINT(ErrorId),0,0);
	16#4310:
		CreateDriveErrMsgDetails := enumMotorEvents.MotorOverTemp ;	
		fnLogMsg(ADR(LogMsg_0),LOG_ERROR,'StepIM Drive ErrorId %d Over-temperature',UDINT_TO_DINT(ErrorId),0,0);
		
	16#5530:
		CreateDriveErrMsgDetails := enumMotorEvents.DriveComError;
		fnLogMsg(ADR(LogMsg_0),LOG_ERROR,'StepIM Drive ErrorId %d EEPROM fault',UDINT_TO_DINT(ErrorId),0,0);
		
	16#7310:
		CreateDriveErrMsgDetails := enumMotorEvents.MotorSpeedError;
		fnLogMsg(ADR(LogMsg_0),LOG_ERROR,'StepIM Drive ErrorId %d Over-speed',UDINT_TO_DINT(ErrorId),0,0);
	16#8130:
		CreateDriveErrMsgDetails := enumMotorEvents.DriveComError;
		fnLogMsg(ADR(LogMsg_0),LOG_ERROR,'StepIM Drive ErrorId %d Heartbeat loss',UDINT_TO_DINT(ErrorId),0,0);
	16#8400:
		CreateDriveErrMsgDetails := enumMotorEvents.MotorSpeedError;
		fnLogMsg(ADR(LogMsg_0),LOG_ERROR,'StepIM Drive ErrorId %d Velocity error',UDINT_TO_DINT(ErrorId),0,0);
	16#8611:
		CreateDriveErrMsgDetails := enumMotorEvents.MotorPositionError;
		fnLogMsg(ADR(LogMsg_0),LOG_ERROR,'StepIM Drive ErrorId %d Position error',UDINT_TO_DINT(ErrorId),0,0);

	16#F001:
 		CreateDriveErrMsgDetails := enumMotorEvents.MotorSpeedError;
		fnLogMsg(ADR(LogMsg_0),LOG_ERROR,'StepIM Drive ErrorId %d Acceleration/deceleration violation',UDINT_TO_DINT(ErrorId),0,0);				
		
	16#FF00: 
		CreateDriveErrMsgDetails := enumMotorEvents.MotorPositionError;
		fnLogMsg(ADR(LogMsg_0),LOG_ERROR,'StepIM Drive ErrorId %d Position Error',UDINT_TO_DINT(ErrorId),0,0);
		
	16#FF03:
		CreateDriveErrMsgDetails := enumMotorEvents.MotorPositionError;
		fnLogMsg(ADR(LogMsg_0),LOG_ERROR,'StepIM Drive ErrorId %d PLL lock lost',UDINT_TO_DINT(ErrorId),0,0);				
		
	16#FF04:
		CreateDriveErrMsgDetails := enumMotorEvents.MotorSupplyError;
		fnLogMsg(ADR(LogMsg_0),LOG_ERROR,'StepIM Drive ErrorId %d Power stage fault',UDINT_TO_DINT(ErrorId),0,0);		
		
	16#FF05:
		CreateDriveErrMsgDetails := enumMotorEvents.MotorFeedBackErr;
		fnLogMsg(ADR(LogMsg_0),LOG_ERROR,'StepIM Drive ErrorId %d Encoder failure',UDINT_TO_DINT(ErrorId),0,0);
	16#FF06:
		CreateDriveErrMsgDetails := enumMotorEvents.MotorSupplyError;
		fnLogMsg(ADR(LogMsg_0),LOG_ERROR,'StepIM Drive ErrorId %d Gate drive voltage Failure',UDINT_TO_DINT(ErrorId),0,0);
	ELSE
		fnLogMsg(ADR(LogMsg_0),LOG_ERROR,'unknown StepIM Drive ErrorId %d ',UDINT_TO_DINT(ErrorId),0,0);
		CreateDriveErrMsgDetails := enumMotorEvents.NoEvents;
END_CASE
END_METHOD

METHOD GetErrCanAdr : BOOL
VAR_INPUT
END_VAR


VAR
	
END_VAR
 SUPER^.GetCanOpenAdr();	

	CoeErrIdIndex	 := 16#603F;
	CoeErrIdSubIndex := 0;
END_METHOD

METHOD  INIT_Specific : BOOL 
VAR_INPUT
	bStart: 					BOOL;
END_VAR
VAR_INST	
	ComDelay:	TON;
	Init_Specific_State : INT ;
	ExecuteTrig: 	Trigger;
END_VAR
IF ExecuteTrig.EDGEPOS(bStart) THEN
	INIT_Specific := FALSE ;
	IF AxisCtrlPtr^.Input.Parameter.Drive.bDisableFoE_Transfer THEN 
		Init_Specific_State:= 4;//10;
	ELSE
		CoEDrive_Ctrl_Adr.ParamsVersionObj.Index    := 16#2F80;
		CoEDrive_Ctrl_Adr.ParamsVersionObj.SunIndex := 1; 		
		Init_Specific_State:= 1;
	END_IF
END_IF


IF ExecuteTrig.EDGENEG(bStart) THEN
	Init_Specific_State := 0;
END_IF	

	
CASE Init_Specific_State OF							
						
	1:	
		Meth_UpdateDriveParams(FALSE);
		Init_Specific_State:=	2;		
	2:
//		SUPER^.ReadInitDriveParID(FALSE);
		IF Meth_UpdateDriveParams(TRUE) THEN
			Init_Specific_State:=	4;
		END_IF	
		

	4:
		
		Init_Specific_State := 0 ;
		INIT_Specific := TRUE ;
		AxisCtrlPtr^.Output.Status.AxisInitDone := TRUE ;
		AxisCtrlPtr^.Output.Status.ReadyForCmd := TRUE ;
END_CASE
END_METHOD

METHOD Meth_CoEChangOperationMode : BOOL
VAR_INPUT
	Execute   : BOOL;	
	OperMode :eCaOpDriveModeOfOperation; 
END_VAR
VAR_INST
	ConfigHomeTrig  : 	Trigger;
	CngOperState : INT;
	Mode      : USINT;	
END_VAR

VAR
	
	
END_VAR
IF ConfigHomeTrig.EDGEPOS(Execute) THEN

	Meth_CoEChangOperationMode := FALSE;				
	Mode := DINT_TO_USINT(OperMode);

	CngOperState := 1;
END_IF


IF ConfigHomeTrig.EDGENEG(Execute) THEN
	
	CngOperState := 0;
END_IF

OperationMode := DINT_TO_USINT(OperMode);
Meth_CoEChangOperationMode := TRUE;
END_METHOD

END_FUNCTION_BLOCK

// ---- POUs/Lib/Motion/ErrorHandling_Lib/FB_ErrorHandler.TcPOU
FUNCTION_BLOCK FINAL FB_ErrorHandler
VAR_INPUT
END_VAR
VAR_OUTPUT
END_VAR
VAR CONSTANT
     EH_MAX_ERROR_ENTRIES  : INT := 30;
END_VAR
VAR
	ErrArr	: ARRAY[0..EH_MAX_ERROR_ENTRIES] OF Eh_ErrorEntry_typ;
	ErrArr_IndexPush	: INT;
	ErrArr_IndexPop		: INT;
	o_IsNotEmpty	: BOOL;
	o_IsEmpty		: BOOL;
	o_IsFull		: BOOL;
	o_IsOverflow	: BOOL;
	o_EntriesCount	: UDINT;
END_VAR

PROPERTY EntriesCount : UDINT
GET
EntriesCount	:= o_EntriesCount;
END_GET
SET
END_SET
END_PROPERTY

METHOD ErrorPop : Eh_ErrorEntry_typ
VAR_INPUT
END_VAR
IF THIS^.o_EntriesCount > 0 THEN
	ErrorPop	:= ErrArr[ErrArr_IndexPop];
	THIS^.o_EntriesCount	:= THIS^.o_EntriesCount - 1;
	ErrArr_IndexPop	:= ErrArr_IndexPop + 1;
	IF THIS^.ErrArr_IndexPop >= EH_MAX_ERROR_ENTRIES THEN
		THIS^.ErrArr_IndexPop	:= 0;
	END_IF
	
	THIS^.o_IsFull		:= FALSE;
	THIS^.o_IsOverflow	:= FALSE;
	IF THIS^.ErrArr_IndexPop = THIS^.ErrArr_IndexPush THEN
		THIS^.o_IsNotEmpty	:= FALSE;
		THIS^.o_IsEmpty		:= TRUE;
	END_IF
END_IF
END_METHOD

METHOD ErrorPush : BOOL
VAR_INPUT
	ErrorEntry	: Eh_ErrorEntry_typ;
END_VAR
IF THIS^.o_EntriesCount < INT_TO_UDINT(EH_MAX_ERROR_ENTRIES) THEN
	// copy data to fifo array
	THIS^.ErrArr[THIS^.ErrArr_IndexPush]	:= ErrorEntry;
	
	// increase push index
	THIS^.ErrArr_IndexPush	:= THIS^.ErrArr_IndexPush + 1;
	IF THIS^.ErrArr_IndexPush >= EH_MAX_ERROR_ENTRIES THEN
		THIS^.ErrArr_IndexPush	:= 0;
	END_IF
	
	// increase entries counter
	THIS^.o_EntriesCount	:= THIS^.o_EntriesCount + 1;
	
	THIS^.o_IsNotEmpty	:= TRUE;
	THIS^.o_IsEmpty		:= FALSE;
	IF THIS^.o_EntriesCount >= INT_TO_UDINT(EH_MAX_ERROR_ENTRIES) THEN
		THIS^.o_IsFull	:= TRUE;
	END_IF
ELSE
	THIS^.o_IsOverflow	:= TRUE;
END_IF
END_METHOD

METHOD ErrorRead : Eh_ErrorEntry_typ
VAR_INPUT
END_VAR
IF THIS^.o_EntriesCount > 0 THEN
	ErrorRead	:= ErrArr[ErrArr_IndexPop];
END_IF
END_METHOD

PROPERTY IsEmpty : BOOL
GET
END_GET
SET
END_SET
END_PROPERTY

PROPERTY IsFull : BOOL
GET
END_GET
SET
END_SET
END_PROPERTY

END_FUNCTION_BLOCK

// ---- POUs/Lib/Motion/EtherCAT/SDO_RW/Tc2_EtherCAT_FB.TcPOU
FUNCTION_BLOCK Tc2_EtherCAT_FB
VAR_INPUT

END_VAR
VAR_OUTPUT
END_VAR
VAR
	ptrTc2_EtherCAT : POINTER TO Tc2_EtherCAT_typ ;
	FB_EcCoeSdoRead_0 	: FB_EcCoeSdoRead ;
	FB_EcCoeSdoWrite_0 	: FB_EcCoeSdoWrite ;
	FB_EcSoeRead_0 		: FB_EcSoeRead ;
	FB_EcSoeWrite_0		: FB_EcSoeWrite ;
	
END_VAR


